LIN {X 0,Y 354.901,Z 540.274,A -85,B 0,C 180,E1 -13338.472,E2 -13338.472} C_VEL
LIN {X 0,Y 354.832,Z 540.28,A -85,B 0,C 180,E1 -13342.106,E2 -13342.106} C_VEL
LIN {X 0,Y 354.892,Z 540.272,A -85,B 0,C 180,E1 -13345.828,E2 -13345.828} C_VEL
LIN {X 0,Y 354.811,Z 540.288,A -85,B 0,C 180,E1 -13349.683,E2 -13349.683} C_VEL
LIN {X 0,Y 354.8,Z 540.289,A -85,B 0,C 180,E1 -13353.703,E2 -13353.703} C_VEL
LIN {X 0,Y 354.793,Z 540.268,A -85,B 0,C 180,E1 -13356.46,E2 -13356.46} C_VEL
LIN {X 0,Y 354.818,Z 540.287,A -85,B 0,C 180,E1 -13359.425,E2 -13359.425} C_VEL
LIN {X 0,Y 354.786,Z 540.277,A -85,B 0,C 180,E1 -13362.869,E2 -13362.869} C_VEL
LIN {X 0,Y 354.836,Z 540.279,A -85,B 0,C 180,E1 -13366.116,E2 -13366.116} C_VEL
LIN {X 0,Y 354.852,Z 540.284,A -85,B 0,C 180,E1 -13369.19,E2 -13369.19} C_VEL
LIN {X 0,Y 354.806,Z 540.261,A -85,B 0,C 180,E1 -13372.403,E2 -13372.403} C_VEL
LIN {X 0,Y 354.81,Z 540.29,A -85,B 0,C 180,E1 -13374.942,E2 -13374.942} C_VEL
LIN {X 0,Y 354.786,Z 540.225,A -85,B 0,C 180,E1 -13378.407,E2 -13378.407} C_VEL
LIN {X 0,Y 354.906,Z 540.442,A -85,B 0,C 180,E1 -13379.59,E2 -13379.59} C_VEL
LIN {X 0,Y 357.393,Z 551.805,A -85,B 0,C 180,E1 -13382.738,E2 -13382.738} C_VEL
LIN {X 0,Y 358.906,Z 560.837,A -85,B 0,C 180,E1 -13385.103,E2 -13385.103} C_VEL
LIN {X 0,Y 357.939,Z 570.577,A -85,B 0,C 180,E1 -13387.413,E2 -13387.413} C_VEL
LIN {X 0,Y 358.417,Z 573.829,A -85,B 0,C 180,E1 -13387.578,E2 -13387.578} C_VEL
LIN {X 0,Y 362.722,Z 599.14,A -85,B 0,C 180,E1 -13388.384,E2 -13388.384} C_VEL
LIN {X 0,Y 363.59,Z 605.924,A -85,B 0,C 180,E1 -13388.579,E2 -13388.579} C_VEL
LIN {X 0,Y 362.337,Z 679.031,A -85,B 0,C 180,E1 -13390.048,E2 -13390.048} C_VEL
LIN {X 0,Y 361.614,Z 692.225,A -85,B 0,C 180,E1 -13390.524,E2 -13390.524} C_VEL
LIN {X 0,Y 360.674,Z 705.472,A -85,B 0,C 180,E1 -13391.247,E2 -13391.247} C_VEL
LIN {X 0,Y 359.694,Z 716.606,A -85,B 0,C 180,E1 -13392.078,E2 -13392.078} C_VEL
LIN {X 0,Y 358.499,Z 728.189,A -85,B 0,C 180,E1 -13393.194,E2 -13393.194} C_VEL
LIN {X 0,Y 357.335,Z 739.084,A -85,B 0,C 180,E1 -13394.521,E2 -13394.521} C_VEL
LIN {X 0,Y 356.269,Z 748.832,A -85,B 0,C 180,E1 -13396.017,E2 -13396.017} C_VEL
LIN {X 0,Y 355.153,Z 757.764,A -85,B 0,C 180,E1 -13397.719,E2 -13397.719} C_VEL
LIN {X 0,Y 354.392,Z 764.959,A -85,B 0,C 180,E1 -13399.431,E2 -13399.431} C_VEL
LIN {X 0,Y 353.9,Z 769.814,A -85,B 0,C 180,E1 -13400.86,E2 -13400.86} C_VEL
LIN {X 0,Y 353.519,Z 774.536,A -85,B 0,C 180,E1 -13402.576,E2 -13402.576} C_VEL
LIN {X 0,Y 353.281,Z 778.149,A -85,B 0,C 180,E1 -13404.293,E2 -13404.293} C_VEL
LIN {X 0,Y 353.28,Z 780.014,A -85,B 0,C 180,E1 -13405.437,E2 -13405.437} C_VEL
LIN {X 0,Y 353.223,Z 781.409,A -85,B 0,C 180,E1 -13406.579,E2 -13406.579} C_VEL
LIN {X 0,Y 353.207,Z 784.384,A -85,B 0,C 180,E1 -13410.001,E2 -13410.001} C_VEL
LIN {X 0,Y 353.167,Z 784.671,A -85,B 0,C 180,E1 -13411.141,E2 -13411.141} C_VEL
LIN {X 0,Y 353.169,Z 784.334,A -85,B 0,C 180,E1 -13412.282,E2 -13412.282} C_VEL
LIN {X 0,Y 353.227,Z 783.434,A -85,B 0,C 180,E1 -13413.423,E2 -13413.423} C_VEL
LIN {X 0,Y 353.326,Z 781.996,A -85,B 0,C 180,E1 -13414.564,E2 -13414.564} C_VEL
LIN {X 0,Y 353.389,Z 779.211,A -85,B 0,C 180,E1 -13416.08,E2 -13416.08} C_VEL
LIN {X 0,Y 353.573,Z 775.814,A -85,B 0,C 180,E1 -13417.424,E2 -13417.424} C_VEL
LIN {X 0,Y 353.842,Z 771.158,A -85,B 0,C 180,E1 -13418.856,E2 -13418.856} C_VEL
LIN {X 0,Y 354.693,Z 761.5,A -85,B 0,C 180,E1 -13421.429,E2 -13421.429} C_VEL
LIN {X 0,Y 355.674,Z 753.468,A -85,B 0,C 180,E1 -13423.135,E2 -13423.135} C_VEL
LIN {X 0,Y 356.598,Z 745.28,A -85,B 0,C 180,E1 -13424.554,E2 -13424.554} C_VEL
LIN {X 0,Y 357.676,Z 735.298,A -85,B 0,C 180,E1 -13425.968,E2 -13425.968} C_VEL
LIN {X 0,Y 358.897,Z 724.022,A -85,B 0,C 180,E1 -13427.229,E2 -13427.229} C_VEL
LIN {X 0,Y 360.015,Z 712.981,A -85,B 0,C 180,E1 -13428.201,E2 -13428.201} C_VEL
LIN {X 0,Y 361.046,Z 700.746,A -85,B 0,C 180,E1 -13429.03,E2 -13429.03} C_VEL
LIN {X 0,Y 361.873,Z 687.862,A -85,B 0,C 180,E1 -13429.648,E2 -13429.648} C_VEL
LIN {X 0,Y 362.44,Z 674.152,A -85,B 0,C 180,E1 -13430.059,E2 -13430.059} C_VEL
LIN {X 0,Y 363.424,Z 603.753,A -85,B 0,C 180,E1 -13431.463,E2 -13431.463} C_VEL
LIN {X 0,Y 360.212,Z 583.434,A -85,B 0,C 180,E1 -13432.106,E2 -13432.106} C_VEL
LIN {X 0,Y 360.059,Z 575.5,A -85,B 0,C 180,E1 -13432.861,E2 -13432.861} C_VEL
LIN {X 0,Y 358.8,Z 563.274,A -85,B 0,C 180,E1 -13434.367,E2 -13434.367} C_VEL
LIN {X 0,Y 358.792,Z 559.513,A -85,B 0,C 180,E1 -13435.217,E2 -13435.217} C_VEL
LIN {X 0,Y 356.679,Z 548.182,A -85,B 0,C 180,E1 -13438.223,E2 -13438.223} C_VEL
LIN {X 0,Y 354.865,Z 540.354,A -85,B 0,C 180,E1 -13440.457,E2 -13440.457} C_VEL
LIN {X 0,Y 354.81,Z 540.287,A -85,B 0,C 180,E1 -13443.702,E2 -13443.702} C_VEL
LIN {X 0,Y 354.802,Z 540.289,A -85,B 0,C 180,E1 -13446.46,E2 -13446.46} C_VEL
LIN {X 0,Y 354.828,Z 540.287,A -85,B 0,C 180,E1 -13449.424,E2 -13449.424} C_VEL
LIN {X 0,Y 354.792,Z 540.29,A -85,B 0,C 180,E1 -13452.868,E2 -13452.868} C_VEL
LIN {X 0,Y 354.77,Z 540.292,A -85,B 0,C 180,E1 -13456.104,E2 -13456.104} C_VEL
LIN {X 0,Y 354.792,Z 540.289,A -85,B 0,C 180,E1 -13459.179,E2 -13459.179} C_VEL
LIN {X 0,Y 354.842,Z 540.398,A -85,B 0,C 180,E1 -13462.926,E2 -13462.926} C_VEL
LIN {X 0,Y 355.958,Z 543.292,A -85,B 0,C 180,E1 -13464.048,E2 -13464.048} C_VEL
LIN {X 0,Y 358.456,Z 549.807,A -85,B 0,C 180,E1 -13466.177,E2 -13466.177} C_VEL
LIN {X 0,Y 361.129,Z 558.129,A -85,B 0,C 180,E1 -13468.551,E2 -13468.551} C_VEL
LIN {X 0,Y 363.277,Z 567.144,A -85,B 0,C 180,E1 -13470.841,E2 -13470.841} C_VEL
LIN {X 0,Y 363.881,Z 571.171,A -85,B 0,C 180,E1 -13471.758,E2 -13471.758} C_VEL
LIN {X 0,Y 362.957,Z 580.6,A -85,B 0,C 180,E1 -13473.554,E2 -13473.554} C_VEL
LIN {X 0,Y 361.094,Z 599.26,A -85,B 0,C 180,E1 -13477.091,E2 -13477.091} C_VEL
LIN {X 0,Y 359.585,Z 617.559,A -85,B 0,C 180,E1 -13480.46,E2 -13480.46} C_VEL
LIN {X 0,Y 362.327,Z 632.262,A -85,B 0,C 180,E1 -13481.252,E2 -13481.252} C_VEL
LIN {X 0,Y 363.24,Z 640.661,A -85,B 0,C 180,E1 -13481.617,E2 -13481.617} C_VEL
LIN {X 0,Y 360.859,Z 699.458,A -85,B 0,C 180,E1 -13483.378,E2 -13483.378} C_VEL
LIN {X 0,Y 360.163,Z 709.923,A -85,B 0,C 180,E1 -13483.855,E2 -13483.855} C_VEL
LIN {X 0,Y 359.446,Z 720.79,A -85,B 0,C 180,E1 -13484.55,E2 -13484.55} C_VEL
LIN {X 0,Y 358.588,Z 730.488,A -85,B 0,C 180,E1 -13485.384,E2 -13485.384} C_VEL
LIN {X 0,Y 357.615,Z 739.515,A -85,B 0,C 180,E1 -13486.36,E2 -13486.36} C_VEL
LIN {X 0,Y 356.754,Z 747.891,A -85,B 0,C 180,E1 -13487.485,E2 -13487.485} C_VEL
LIN {X 0,Y 355.858,Z 756.225,A -85,B 0,C 180,E1 -13488.898,E2 -13488.898} C_VEL
LIN {X 0,Y 355.005,Z 762.802,A -85,B 0,C 180,E1 -13490.313,E2 -13490.313} C_VEL
LIN {X 0,Y 354.501,Z 767.137,A -85,B 0,C 180,E1 -13491.449,E2 -13491.449} C_VEL
LIN {X 0,Y 354.019,Z 771.909,A -85,B 0,C 180,E1 -13493.031,E2 -13493.031} C_VEL
LIN {X 0,Y 353.804,Z 774.792,A -85,B 0,C 180,E1 -13494.3,E2 -13494.3} C_VEL
LIN {X 0,Y 353.489,Z 776.752,A -85,B 0,C 180,E1 -13495.439,E2 -13495.439} C_VEL
LIN {X 0,Y 353.296,Z 778.158,A -85,B 0,C 180,E1 -13496.579,E2 -13496.579} C_VEL
LIN {X 0,Y 353.211,Z 779.033,A -85,B 0,C 180,E1 -13497.719,E2 -13497.719} C_VEL
LIN {X 0,Y 353.165,Z 779.34,A -85,B 0,C 180,E1 -13498.86,E2 -13498.86} C_VEL
LIN {X 0,Y 353.174,Z 779.041,A -85,B 0,C 180,E1 -13500,E2 -13500} C_VEL
LIN {X 0,Y 353.158,Z 778.209,A -85,B 0,C 180,E1 -13501.14,E2 -13501.14} C_VEL
LIN {X 0,Y 353.181,Z 776.838,A -85,B 0,C 180,E1 -13502.281,E2 -13502.281} C_VEL
LIN {X 0,Y 353.348,Z 773.707,A -85,B 0,C 180,E1 -13503.992,E2 -13503.992} C_VEL
LIN {X 0,Y 353.451,Z 769.159,A -85,B 0,C 180,E1 -13505.706,E2 -13505.706} C_VEL
LIN {X 0,Y 353.752,Z 764.04,A -85,B 0,C 180,E1 -13507.133,E2 -13507.133} C_VEL
LIN {X 0,Y 353.938,Z 759.008,A -85,B 0,C 180,E1 -13508.277,E2 -13508.277} C_VEL
LIN {X 0,Y 354.29,Z 752.942,A -85,B 0,C 180,E1 -13509.419,E2 -13509.419} C_VEL
LIN {X 0,Y 354.719,Z 745.593,A -85,B 0,C 180,E1 -13510.56,E2 -13510.56} C_VEL
LIN {X 0,Y 355.216,Z 736.599,A -85,B 0,C 180,E1 -13511.701,E2 -13511.701} C_VEL
LIN {X 0,Y 355.821,Z 726.511,A -85,B 0,C 180,E1 -13512.694,E2 -13512.694} C_VEL
LIN {X 0,Y 356.24,Z 717.243,A -85,B 0,C 180,E1 -13513.404,E2 -13513.404} C_VEL
LIN {X 0,Y 356.538,Z 707.589,A -85,B 0,C 180,E1 -13513.973,E2 -13513.973} C_VEL
LIN {X 0,Y 356.953,Z 695.613,A -85,B 0,C 180,E1 -13514.466,E2 -13514.466} C_VEL
LIN {X 0,Y 357.953,Z 636.557,A -85,B 0,C 180,E1 -13516.028,E2 -13516.028} C_VEL
LIN {X 0,Y 356.048,Z 617.144,A -85,B 0,C 180,E1 -13516.632,E2 -13516.632} C_VEL
LIN {X 0,Y 356.832,Z 600.704,A -85,B 0,C 180,E1 -13519.562,E2 -13519.562} C_VEL
LIN {X 0,Y 358.029,Z 581.082,A -85,B 0,C 180,E1 -13523.116,E2 -13523.116} C_VEL
LIN {X 0,Y 359.095,Z 562.902,A -85,B 0,C 180,E1 -13526.425,E2 -13526.425} C_VEL
LIN {X 0,Y 358.505,Z 557.641,A -85,B 0,C 180,E1 -13527.429,E2 -13527.429} C_VEL
LIN {X 0,Y 355.305,Z 542.619,A -85,B 0,C 180,E1 -13530.406,E2 -13530.406} C_VEL
LIN {X 0,Y 354.856,Z 540.394,A -85,B 0,C 180,E1 -13530.902,E2 -13530.902} C_VEL
LIN {X 0,Y 354.816,Z 540.289,A -85,B 0,C 180,E1 -13535.059,E2 -13535.059} C_VEL
LIN {X 0,Y 354.814,Z 540.286,A -85,B 0,C 180,E1 -13537.882,E2 -13537.882} C_VEL
LIN {X 0,Y 354.79,Z 540.253,A -85,B 0,C 180,E1 -13541.171,E2 -13541.171} C_VEL
LIN {X 0,Y 354.767,Z 540.28,A -85,B 0,C 180,E1 -13544.506,E2 -13544.506} C_VEL
LIN {X 0,Y 354.798,Z 540.285,A -85,B 0,C 180,E1 -13547.662,E2 -13547.662} C_VEL
LIN {X 0,Y 354.819,Z 540.256,A -85,B 0,C 180,E1 -13550.666,E2 -13550.666} C_VEL
LIN {X 0,Y 354.826,Z 540.285,A -85,B 0,C 180,E1 -13554.3,E2 -13554.3} C_VEL
LIN {X 0,Y 354.791,Z 540.29,A -85,B 0,C 180,E1 -13557.666,E2 -13557.666} C_VEL
LIN {X 0,Y 354.851,Z 540.28,A -85,B 0,C 180,E1 -13561.618,E2 -13561.618} C_VEL
LIN {X 0,Y 354.938,Z 540.423,A -85,B 0,C 180,E1 -13563.859,E2 -13563.859} C_VEL
LIN {X 0,Y 356.824,Z 549.951,A -85,B 0,C 180,E1 -13566.801,E2 -13566.801} C_VEL
LIN {X 0,Y 357.319,Z 552.539,A -85,B 0,C 180,E1 -13567.484,E2 -13567.484} C_VEL
LIN {X 0,Y 360.175,Z 560.7,A -85,B 0,C 180,E1 -13567.881,E2 -13567.881} C_VEL
LIN {X 0,Y 363.978,Z 579.583,A -85,B 0,C 180,E1 -13568.52,E2 -13568.52} C_VEL
LIN {X 0,Y 362.543,Z 658.643,A -85,B 0,C 180,E1 -13570.095,E2 -13570.095} C_VEL
LIN {X 0,Y 362.059,Z 671.327,A -85,B 0,C 180,E1 -13570.547,E2 -13570.547} C_VEL
LIN {X 0,Y 361.211,Z 684.868,A -85,B 0,C 180,E1 -13571.274,E2 -13571.274} C_VEL
LIN {X 0,Y 360.315,Z 696.202,A -85,B 0,C 180,E1 -13572.108,E2 -13572.108} C_VEL
LIN {X 0,Y 359.184,Z 707.773,A -85,B 0,C 180,E1 -13573.215,E2 -13573.215} C_VEL
LIN {X 0,Y 358.249,Z 718.308,A -85,B 0,C 180,E1 -13574.496,E2 -13574.496} C_VEL
LIN {X 0,Y 357.199,Z 726.851,A -85,B 0,C 180,E1 -13575.762,E2 -13575.762} C_VEL
LIN {X 0,Y 356.221,Z 734.721,A -85,B 0,C 180,E1 -13577.175,E2 -13577.175} C_VEL
LIN {X 0,Y 355.29,Z 742.41,A -85,B 0,C 180,E1 -13578.879,E2 -13578.879} C_VEL
LIN {X 0,Y 354.406,Z 749.468,A -85,B 0,C 180,E1 -13580.871,E2 -13580.871} C_VEL
LIN {X 0,Y 353.946,Z 754.166,A -85,B 0,C 180,E1 -13582.584,E2 -13582.584} C_VEL
LIN {X 0,Y 353.676,Z 757.756,A -85,B 0,C 180,E1 -13584.297,E2 -13584.297} C_VEL
LIN {X 0,Y 353.497,Z 759.613,A -85,B 0,C 180,E1 -13585.438,E2 -13585.438} C_VEL
LIN {X 0,Y 353.34,Z 761.013,A -85,B 0,C 180,E1 -13586.578,E2 -13586.578} C_VEL
LIN {X 0,Y 353.256,Z 762.621,A -85,B 0,C 180,E1 -13588.859,E2 -13588.859} C_VEL
LIN {X 0,Y 353.265,Z 762.853,A -85,B 0,C 180,E1 -13589.999,E2 -13589.999} C_VEL
LIN {X 0,Y 353.256,Z 762.665,A -85,B 0,C 180,E1 -13591.139,E2 -13591.139} C_VEL
LIN {X 0,Y 353.334,Z 761.117,A -85,B 0,C 180,E1 -13593.42,E2 -13593.42} C_VEL
LIN {X 0,Y 353.49,Z 759.761,A -85,B 0,C 180,E1 -13594.56,E2 -13594.56} C_VEL
LIN {X 0,Y 353.814,Z 756.019,A -85,B 0,C 180,E1 -13596.695,E2 -13596.695} C_VEL
LIN {X 0,Y 354.2,Z 751.45,A -85,B 0,C 180,E1 -13598.557,E2 -13598.557} C_VEL
LIN {X 0,Y 355.015,Z 745.015,A -85,B 0,C 180,E1 -13600.55,E2 -13600.55} C_VEL
LIN {X 0,Y 355.74,Z 738.678,A -85,B 0,C 180,E1 -13602.095,E2 -13602.095} C_VEL
LIN {X 0,Y 355.481,Z 735.193,A -85,B 0,C 180,E1 -13602.864,E2 -13602.864} C_VEL
LIN {X 0,Y 353.491,Z 729.249,A -85,B 0,C 180,E1 -13604.108,E2 -13604.108} C_VEL
LIN {X 0,Y 351.566,Z 722.759,A -85,B 0,C 180,E1 -13605.284,E2 -13605.284} C_VEL
LIN {X 0,Y 351.399,Z 718.404,A -85,B 0,C 180,E1 -13605.933,E2 -13605.933} C_VEL
LIN {X 0,Y 352.412,Z 707.819,A -85,B 0,C 180,E1 -13607.24,E2 -13607.24} C_VEL
LIN {X 0,Y 353.608,Z 695.92,A -85,B 0,C 180,E1 -13608.391,E2 -13608.391} C_VEL
LIN {X 0,Y 354.725,Z 683.279,A -85,B 0,C 180,E1 -13609.305,E2 -13609.305} C_VEL
LIN {X 0,Y 355.479,Z 670.635,A -85,B 0,C 180,E1 -13609.977,E2 -13609.977} C_VEL
LIN {X 0,Y 355.945,Z 658.621,A -85,B 0,C 180,E1 -13610.401,E2 -13610.401} C_VEL
LIN {X 0,Y 357.347,Z 579.911,A -85,B 0,C 180,E1 -13612.002,E2 -13612.002} C_VEL
LIN {X 0,Y 353.421,Z 561.513,A -85,B 0,C 180,E1 -13612.658,E2 -13612.658} C_VEL
LIN {X 0,Y 350.203,Z 552.682,A -85,B 0,C 180,E1 -13613.115,E2 -13613.115} C_VEL
LIN {X 0,Y 348.907,Z 546.369,A -85,B 0,C 180,E1 -13614.983,E2 -13614.983} C_VEL
LIN {X 0,Y 347.866,Z 541.204,A -85,B 0,C 180,E1 -13616.687,E2 -13616.687} C_VEL
LIN {X 0,Y 347.747,Z 541.157,A -85,B 0,C 180,E1 -13620.347,E2 -13620.347} C_VEL
LIN {X 0,Y 347.746,Z 541.17,A -85,B 0,C 180,E1 -13624.043,E2 -13624.043} C_VEL
LIN {X 0,Y 347.763,Z 541.166,A -85,B 0,C 180,E1 -13627.319,E2 -13627.319} C_VEL
LIN {X 0,Y 347.74,Z 541.16,A -85,B 0,C 180,E1 -13630.294,E2 -13630.294} C_VEL
LIN {X 0,Y 347.72,Z 541.166,A -85,B 0,C 180,E1 -13633.407,E2 -13633.407} C_VEL
LIN {X 0,Y 347.742,Z 541.163,A -85,B 0,C 180,E1 -13636.681,E2 -13636.681} C_VEL
LIN {X 0,Y 347.753,Z 541.153,A -85,B 0,C 180,E1 -13640.17,E2 -13640.17} C_VEL
LIN {X 0,Y 347.762,Z 541.151,A -85,B 0,C 180,E1 -13642.679,E2 -13642.679} C_VEL
LIN {X 0,Y 347.743,Z 541.167,A -85,B 0,C 180,E1 -13645.955,E2 -13645.955} C_VEL
LIN {X 0,Y 347.758,Z 541.169,A -85,B 0,C 180,E1 -13649.653,E2 -13649.653} C_VEL
LIN {X 0,Y 347.846,Z 541.145,A -85,B 0,C 180,E1 -13652.744,E2 -13652.744} C_VEL
LIN {X 0,Y 347.782,Z 541.159,A -85,B 0,C 180,E1 -13656.161,E2 -13656.161} C_VEL
LIN {X 0,Y 347.811,Z 541.159,A -85,B 0,C 180,E1 -13659.909,E2 -13659.909} C_VEL
LIN {X 0,Y 347.859,Z 541.147,A -85,B 0,C 180,E1 -13662.359,E2 -13662.359} C_VEL
LIN {X 0,Y 347.89,Z 541.149,A -85,B 0,C 180,E1 -13665.97,E2 -13665.97} C_VEL
LIN {X 0,Y 347.921,Z 541.135,A -85,B 0,C 180,E1 -13669.525,E2 -13669.525} C_VEL
LIN {X 0,Y 348.067,Z 541.126,A -85,B 0,C 180,E1 -13671.874,E2 -13671.874} C_VEL
LIN {X 0,Y 348.06,Z 541.126,A -85,B 0,C 180,E1 -13674.205,E2 -13674.205} C_VEL
LIN {X 0,Y 348.201,Z 541.102,A -85,B 0,C 180,E1 -13677.686,E2 -13677.686} C_VEL
LIN {X 0,Y 348.361,Z 541.091,A -85,B 0,C 180,E1 -13680,E2 -13680} C_VEL
LIN {X 0,Y 348.201,Z 541.103,A -85,B 0,C 180,E1 -13682.313,E2 -13682.313} C_VEL
LIN {X 0,Y 348.101,Z 541.122,A -85,B 0,C 180,E1 -13686.958,E2 -13686.958} C_VEL
LIN {X 0,Y 347.961,Z 541.134,A -85,B 0,C 180,E1 -13689.299,E2 -13689.299} C_VEL
LIN {X 0,Y 347.886,Z 541.148,A -85,B 0,C 180,E1 -13692.84,E2 -13692.84} C_VEL
LIN {X 0,Y 347.832,Z 541.147,A -85,B 0,C 180,E1 -13696.432,E2 -13696.432} C_VEL
LIN {X 0,Y 347.852,Z 541.153,A -85,B 0,C 180,E1 -13698.86,E2 -13698.86} C_VEL
LIN {X 0,Y 347.77,Z 541.159,A -85,B 0,C 180,E1 -13702.58,E2 -13702.58} C_VEL
LIN {X 0,Y 347.806,Z 541.16,A -85,B 0,C 180,E1 -13705.109,E2 -13705.109} C_VEL
LIN {X 0,Y 347.801,Z 541.158,A -85,B 0,C 180,E1 -13707.695,E2 -13707.695} C_VEL
LIN {X 0,Y 347.743,Z 541.163,A -85,B 0,C 180,E1 -13710.349,E2 -13710.349} C_VEL
LIN {X 0,Y 347.742,Z 541.165,A -85,B 0,C 180,E1 -13714.045,E2 -13714.045} C_VEL
LIN {X 0,Y 347.757,Z 541.148,A -85,B 0,C 180,E1 -13717.322,E2 -13717.322} C_VEL
LIN {X 0,Y 347.728,Z 541.169,A -85,B 0,C 180,E1 -13720.298,E2 -13720.298} C_VEL
LIN {X 0,Y 347.742,Z 541.158,A -85,B 0,C 180,E1 -13723.405,E2 -13723.405} C_VEL
LIN {X 0,Y 347.778,Z 541.155,A -85,B 0,C 180,E1 -13726.677,E2 -13726.677} C_VEL
LIN {X 0,Y 347.782,Z 541.157,A -85,B 0,C 180,E1 -13730.166,E2 -13730.166} C_VEL
LIN {X 0,Y 347.786,Z 541.158,A -85,B 0,C 180,E1 -13734.126,E2 -13734.126} C_VEL
LIN {X 0,Y 347.732,Z 541.104,A -85,B 0,C 180,E1 -13738.088,E2 -13738.088} C_VEL
LIN {X 0,Y 347.806,Z 541.332,A -85,B 0,C 180,E1 -13739.197,E2 -13739.197} C_VEL
LIN {X 0,Y 350.44,Z 553.084,A -85,B 0,C 180,E1 -13742.533,E2 -13742.533} C_VEL
LIN {X 0,Y 351.969,Z 561.98,A -85,B 0,C 180,E1 -13744.92,E2 -13744.92} C_VEL
LIN {X 0,Y 351.14,Z 570.571,A -85,B 0,C 180,E1 -13746.977,E2 -13746.977} C_VEL
LIN {X 0,Y 352.793,Z 579.779,A -85,B 0,C 180,E1 -13747.333,E2 -13747.333} C_VEL
LIN {X 0,Y 356.961,Z 605.801,A -85,B 0,C 180,E1 -13748.162,E2 -13748.162} C_VEL
LIN {X 0,Y 355.687,Z 678.839,A -85,B 0,C 180,E1 -13749.659,E2 -13749.659} C_VEL
LIN {X 0,Y 354.941,Z 692.03,A -85,B 0,C 180,E1 -13750.142,E2 -13750.142} C_VEL
LIN {X 0,Y 353.972,Z 705.273,A -85,B 0,C 180,E1 -13750.878,E2 -13750.878} C_VEL
LIN {X 0,Y 352.931,Z 716.405,A -85,B 0,C 180,E1 -13751.723,E2 -13751.723} C_VEL
LIN {X 0,Y 351.685,Z 727.987,A -85,B 0,C 180,E1 -13752.858,E2 -13752.858} C_VEL
LIN {X 0,Y 350.454,Z 738.96,A -85,B 0,C 180,E1 -13754.22,E2 -13754.22} C_VEL
LIN {X 0,Y 349.343,Z 748.628,A -85,B 0,C 180,E1 -13755.734,E2 -13755.734} C_VEL
LIN {X 0,Y 348.199,Z 757.561,A -85,B 0,C 180,E1 -13757.47,E2 -13757.47} C_VEL
LIN {X 0,Y 347.398,Z 764.755,A -85,B 0,C 180,E1 -13759.216,E2 -13759.216} C_VEL
LIN {X 0,Y 346.719,Z 771.305,A -85,B 0,C 180,E1 -13761.257,E2 -13761.257} C_VEL
LIN {X 0,Y 346.343,Z 775.644,A -85,B 0,C 180,E1 -13763.008,E2 -13763.008} C_VEL
LIN {X 0,Y 346.2,Z 777.944,A -85,B 0,C 180,E1 -13764.175,E2 -13764.175} C_VEL
LIN {X 0,Y 346.175,Z 779.809,A -85,B 0,C 180,E1 -13765.343,E2 -13765.343} C_VEL
LIN {X 0,Y 346.147,Z 781.205,A -85,B 0,C 180,E1 -13766.509,E2 -13766.509} C_VEL
LIN {X 0,Y 346.108,Z 784.272,A -85,B 0,C 180,E1 -13770.001,E2 -13770.001} C_VEL
LIN {X 0,Y 346.069,Z 784.599,A -85,B 0,C 180,E1 -13771.165,E2 -13771.165} C_VEL
LIN {X 0,Y 346.081,Z 784.321,A -85,B 0,C 180,E1 -13772.329,E2 -13772.329} C_VEL
LIN {X 0,Y 346.154,Z 783.509,A -85,B 0,C 180,E1 -13773.493,E2 -13773.493} C_VEL
LIN {X 0,Y 346.239,Z 782.157,A -85,B 0,C 180,E1 -13774.658,E2 -13774.658} C_VEL
LIN {X 0,Y 346.326,Z 779.703,A -85,B 0,C 180,E1 -13776.087,E2 -13776.087} C_VEL
LIN {X 0,Y 346.545,Z 776.182,A -85,B 0,C 180,E1 -13777.576,E2 -13777.576} C_VEL
LIN {X 0,Y 346.788,Z 772.656,A -85,B 0,C 180,E1 -13778.743,E2 -13778.743} C_VEL
LIN {X 0,Y 347.163,Z 767.179,A -85,B 0,C 180,E1 -13780.204,E2 -13780.204} C_VEL
LIN {X 0,Y 348.199,Z 757.494,A -85,B 0,C 180,E1 -13782.532,E2 -13782.532} C_VEL
LIN {X 0,Y 349.322,Z 748.545,A -85,B 0,C 180,E1 -13784.269,E2 -13784.269} C_VEL
LIN {X 0,Y 350.431,Z 738.64,A -85,B 0,C 180,E1 -13785.813,E2 -13785.813} C_VEL
LIN {X 0,Y 351.633,Z 727.851,A -85,B 0,C 180,E1 -13787.147,E2 -13787.147} C_VEL
LIN {X 0,Y 352.906,Z 716.238,A -85,B 0,C 180,E1 -13788.281,E2 -13788.281} C_VEL
LIN {X 0,Y 354.038,Z 703.927,A -85,B 0,C 180,E1 -13789.196,E2 -13789.196} C_VEL
LIN {X 0,Y 354.969,Z 690.954,A -85,B 0,C 180,E1 -13789.896,E2 -13789.896} C_VEL
LIN {X 0,Y 355.681,Z 678.349,A -85,B 0,C 180,E1 -13790.344,E2 -13790.344} C_VEL
LIN {X 0,Y 356.835,Z 604.804,A -85,B 0,C 180,E1 -13791.852,E2 -13791.852} C_VEL
LIN {X 0,Y 354.448,Z 588.941,A -85,B 0,C 180,E1 -13792.364,E2 -13792.364} C_VEL
LIN {X 0,Y 354.5,Z 578.627,A -85,B 0,C 180,E1 -13793.361,E2 -13793.361} C_VEL
LIN {X 0,Y 353.313,Z 565.845,A -85,B 0,C 180,E1 -13794.979,E2 -13794.979} C_VEL
LIN {X 0,Y 351.074,Z 556.144,A -85,B 0,C 180,E1 -13796.711,E2 -13796.711} C_VEL
LIN {X 0,Y 349.591,Z 548.971,A -85,B 0,C 180,E1 -13798.587,E2 -13798.587} C_VEL
LIN {X 0,Y 347.804,Z 541.258,A -85,B 0,C 180,E1 -13800.848,E2 -13800.848} C_VEL
LIN {X 0,Y 347.748,Z 541.169,A -85,B 0,C 180,E1 -13804.464,E2 -13804.464} C_VEL
LIN {X 0,Y 347.777,Z 541.166,A -85,B 0,C 180,E1 -13807.989,E2 -13807.989} C_VEL
LIN {X 0,Y 347.754,Z 541.167,A -85,B 0,C 180,E1 -13811.831,E2 -13811.831} C_VEL
LIN {X 0,Y 347.709,Z 541.175,A -85,B 0,C 180,E1 -13815.027,E2 -13815.027} C_VEL
LIN {X 0,Y 347.754,Z 541.168,A -85,B 0,C 180,E1 -13818.398,E2 -13818.398} C_VEL
LIN {X 0,Y 347.787,Z 541.37,A -85,B 0,C 180,E1 -13821.325,E2 -13821.325} C_VEL
LIN {X 0,Y 348.698,Z 543.886,A -85,B 0,C 180,E1 -13822.392,E2 -13822.392} C_VEL
LIN {X 0,Y 349.391,Z 544.951,A -85,B 0,C 180,E1 -13822.883,E2 -13822.883} C_VEL
LIN {X 0,Y 352.197,Z 552.266,A -85,B 0,C 180,E1 -13825.492,E2 -13825.492} C_VEL
LIN {X 0,Y 354.798,Z 560.426,A -85,B 0,C 180,E1 -13827.979,E2 -13827.979} C_VEL
LIN {X 0,Y 356.732,Z 568.33,A -85,B 0,C 180,E1 -13830.095,E2 -13830.095} C_VEL
LIN {X 0,Y 357.593,Z 574.274,A -85,B 0,C 180,E1 -13831.536,E2 -13831.536} C_VEL
LIN {X 0,Y 355.71,Z 591.496,A -85,B 0,C 180,E1 -13834.863,E2 -13834.863} C_VEL
LIN {X 0,Y 353.484,Z 613.273,A -85,B 0,C 180,E1 -13839.03,E2 -13839.03} C_VEL
LIN {X 0,Y 353.182,Z 617.698,A -85,B 0,C 180,E1 -13839.815,E2 -13839.815} C_VEL
LIN {X 0,Y 356.187,Z 633.43,A -85,B 0,C 180,E1 -13840.71,E2 -13840.71} C_VEL
LIN {X 0,Y 357.042,Z 641.425,A -85,B 0,C 180,E1 -13841.084,E2 -13841.084} C_VEL
LIN {X 0,Y 354.464,Z 699.698,A -85,B 0,C 180,E1 -13842.884,E2 -13842.884} C_VEL
LIN {X 0,Y 353.79,Z 709.378,A -85,B 0,C 180,E1 -13843.334,E2 -13843.334} C_VEL
LIN {X 0,Y 352.925,Z 721.212,A -85,B 0,C 180,E1 -13844.109,E2 -13844.109} C_VEL
LIN {X 0,Y 351.981,Z 730.75,A -85,B 0,C 180,E1 -13844.955,E2 -13844.955} C_VEL
LIN {X 0,Y 350.956,Z 739.685,A -85,B 0,C 180,E1 -13845.948,E2 -13845.948} C_VEL
LIN {X 0,Y 350.109,Z 747.08,A -85,B 0,C 180,E1 -13846.948,E2 -13846.948} C_VEL
LIN {X 0,Y 349.148,Z 755.674,A -85,B 0,C 180,E1 -13848.388,E2 -13848.388} C_VEL
LIN {X 0,Y 348.212,Z 762.369,A -85,B 0,C 180,E1 -13849.828,E2 -13849.828} C_VEL
LIN {X 0,Y 347.524,Z 767.736,A -85,B 0,C 180,E1 -13851.276,E2 -13851.276} C_VEL
LIN {X 0,Y 347.123,Z 771.195,A -85,B 0,C 180,E1 -13852.438,E2 -13852.438} C_VEL
LIN {X 0,Y 346.766,Z 775.162,A -85,B 0,C 180,E1 -13854.184,E2 -13854.184} C_VEL
LIN {X 0,Y 346.439,Z 777.035,A -85,B 0,C 180,E1 -13855.346,E2 -13855.346} C_VEL
LIN {X 0,Y 346.224,Z 778.353,A -85,B 0,C 180,E1 -13856.509,E2 -13856.509} C_VEL
LIN {X 0,Y 346.123,Z 779.14,A -85,B 0,C 180,E1 -13857.673,E2 -13857.673} C_VEL
LIN {X 0,Y 346.068,Z 779.396,A -85,B 0,C 180,E1 -13858.836,E2 -13858.836} C_VEL
LIN {X 0,Y 346.074,Z 779.051,A -85,B 0,C 180,E1 -13860,E2 -13860} C_VEL
LIN {X 0,Y 346.061,Z 778.124,A -85,B 0,C 180,E1 -13861.164,E2 -13861.164} C_VEL
LIN {X 0,Y 346.127,Z 775.788,A -85,B 0,C 180,E1 -13862.91,E2 -13862.91} C_VEL
LIN {X 0,Y 346.314,Z 771.991,A -85,B 0,C 180,E1 -13864.656,E2 -13864.656} C_VEL
LIN {X 0,Y 346.45,Z 767.166,A -85,B 0,C 180,E1 -13866.274,E2 -13866.274} C_VEL
LIN {X 0,Y 346.778,Z 761.051,A -85,B 0,C 180,E1 -13867.863,E2 -13867.863} C_VEL
LIN {X 0,Y 347.173,Z 753.767,A -85,B 0,C 180,E1 -13869.32,E2 -13869.32} C_VEL
LIN {X 0,Y 347.643,Z 745.538,A -85,B 0,C 180,E1 -13870.63,E2 -13870.63} C_VEL
LIN {X 0,Y 348.149,Z 736.517,A -85,B 0,C 180,E1 -13871.794,E2 -13871.794} C_VEL
LIN {X 0,Y 348.779,Z 726.368,A -85,B 0,C 180,E1 -13872.806,E2 -13872.806} C_VEL
LIN {X 0,Y 349.201,Z 717.059,A -85,B 0,C 180,E1 -13873.531,E2 -13873.531} C_VEL
LIN {X 0,Y 349.497,Z 707.355,A -85,B 0,C 180,E1 -13874.112,E2 -13874.112} C_VEL
LIN {X 0,Y 349.934,Z 695.198,A -85,B 0,C 180,E1 -13874.614,E2 -13874.614} C_VEL
LIN {X 0,Y 350.971,Z 637.15,A -85,B 0,C 180,E1 -13876.193,E2 -13876.193} C_VEL
LIN {X 0,Y 349.033,Z 617.196,A -85,B 0,C 180,E1 -13876.825,E2 -13876.825} C_VEL
LIN {X 0,Y 349.811,Z 601.182,A -85,B 0,C 180,E1 -13879.719,E2 -13879.719} C_VEL
LIN {X 0,Y 351.07,Z 581.28,A -85,B 0,C 180,E1 -13883.375,E2 -13883.375} C_VEL
LIN {X 0,Y 352.127,Z 563.318,A -85,B 0,C 180,E1 -13886.684,E2 -13886.684} C_VEL
LIN {X 0,Y 350.727,Z 554.833,A -85,B 0,C 180,E1 -13888.353,E2 -13888.353} C_VEL
LIN {X 0,Y 347.808,Z 541.27,A -85,B 0,C 180,E1 -13891.142,E2 -13891.142} C_VEL
LIN {X 0,Y 347.748,Z 541.168,A -85,B 0,C 180,E1 -13894.464,E2 -13894.464} C_VEL
LIN {X 0,Y 347.781,Z 541.162,A -85,B 0,C 180,E1 -13897.989,E2 -13897.989} C_VEL
LIN {X 0,Y 347.754,Z 541.122,A -85,B 0,C 180,E1 -13901.83,E2 -13901.83} C_VEL
LIN {X 0,Y 347.71,Z 541.162,A -85,B 0,C 180,E1 -13905.026,E2 -13905.026} C_VEL
LIN {X 0,Y 347.754,Z 541.157,A -85,B 0,C 180,E1 -13908.397,E2 -13908.397} C_VEL
LIN {X 0,Y 347.777,Z 541.152,A -85,B 0,C 180,E1 -13912.011,E2 -13912.011} C_VEL
LIN {X 0,Y 347.748,Z 541.158,A -85,B 0,C 180,E1 -13915.536,E2 -13915.536} C_VEL
LIN {X 0,Y 347.749,Z 541.164,A -85,B 0,C 180,E1 -13918.3,E2 -13918.3} C_VEL
LIN {X 0,Y 347.783,Z 541.162,A -85,B 0,C 180,E1 -13920.987,E2 -13920.987} C_VEL
LIN {X 0,Y 347.898,Z 541.271,A -85,B 0,C 180,E1 -13923.48,E2 -13923.48} C_VEL
LIN {X 0,Y 349.965,Z 551.705,A -85,B 0,C 180,E1 -13926.765,E2 -13926.765} C_VEL
LIN {X 0,Y 350.215,Z 552.951,A -85,B 0,C 180,E1 -13927.018,E2 -13927.018} C_VEL
LIN {X 0,Y 353.926,Z 563.388,A -85,B 0,C 180,E1 -13927.522,E2 -13927.522} C_VEL
LIN {X 0,Y 357.382,Z 580.666,A -85,B 0,C 180,E1 -13928.121,E2 -13928.121} C_VEL
LIN {X 0,Y 355.903,Z 658.865,A -85,B 0,C 180,E1 -13929.707,E2 -13929.707} C_VEL
LIN {X 0,Y 355.396,Z 671.542,A -85,B 0,C 180,E1 -13930.167,E2 -13930.167} C_VEL
LIN {X 0,Y 354.517,Z 685.08,A -85,B 0,C 180,E1 -13930.906,E2 -13930.906} C_VEL
LIN {X 0,Y 353.579,Z 696.412,A -85,B 0,C 180,E1 -13931.755,E2 -13931.755} C_VEL
LIN {X 0,Y 352.368,Z 708.321,A -85,B 0,C 180,E1 -13932.92,E2 -13932.92} C_VEL
LIN {X 0,Y 351.411,Z 718.516,A -85,B 0,C 180,E1 -13934.187,E2 -13934.187} C_VEL
LIN {X 0,Y 350.321,Z 727.059,A -85,B 0,C 180,E1 -13935.476,E2 -13935.476} C_VEL
LIN {X 0,Y 349.282,Z 734.929,A -85,B 0,C 180,E1 -13936.916,E2 -13936.916} C_VEL
LIN {X 0,Y 348.321,Z 742.616,A -85,B 0,C 180,E1 -13938.654,E2 -13938.654} C_VEL
LIN {X 0,Y 347.656,Z 747.865,A -85,B 0,C 180,E1 -13940.105,E2 -13940.105} C_VEL
LIN {X 0,Y 347.019,Z 752.957,A -85,B 0,C 180,E1 -13941.849,E2 -13941.849} C_VEL
LIN {X 0,Y 346.728,Z 756.326,A -85,B 0,C 180,E1 -13943.32,E2 -13943.32} C_VEL
LIN {X 0,Y 346.439,Z 759.818,A -85,B 0,C 180,E1 -13945.345,E2 -13945.345} C_VEL
LIN {X 0,Y 346.264,Z 761.218,A -85,B 0,C 180,E1 -13946.508,E2 -13946.508} C_VEL
LIN {X 0,Y 346.16,Z 762.826,A -85,B 0,C 180,E1 -13948.836,E2 -13948.836} C_VEL
LIN {X 0,Y 346.168,Z 763.058,A -85,B 0,C 180,E1 -13949.999,E2 -13949.999} C_VEL
LIN {X 0,Y 346.159,Z 762.869,A -85,B 0,C 180,E1 -13951.162,E2 -13951.162} C_VEL
LIN {X 0,Y 346.259,Z 761.321,A -85,B 0,C 180,E1 -13953.49,E2 -13953.49} C_VEL
LIN {X 0,Y 346.432,Z 759.964,A -85,B 0,C 180,E1 -13954.653,E2 -13954.653} C_VEL
LIN {X 0,Y 346.727,Z 756.547,A -85,B 0,C 180,E1 -13956.679,E2 -13956.679} C_VEL
LIN {X 0,Y 347.175,Z 751.654,A -85,B 0,C 180,E1 -13958.732,E2 -13958.732} C_VEL
LIN {X 0,Y 348.004,Z 745.219,A -85,B 0,C 180,E1 -13960.765,E2 -13960.765} C_VEL
LIN {X 0,Y 348.861,Z 738.146,A -85,B 0,C 180,E1 -13962.506,E2 -13962.506} C_VEL
LIN {X 0,Y 350.045,Z 729.329,A -85,B 0,C 180,E1 -13964.237,E2 -13964.237} C_VEL
LIN {X 0,Y 351.213,Z 720.287,A -85,B 0,C 180,E1 -13965.67,E2 -13965.67} C_VEL
LIN {X 0,Y 351.399,Z 718.404,A -85,B 0,C 180,E1 -13965.933,E2 -13965.933} C_VEL
LIN {X 0,Y 351.194,Z 713.945,A -85,B 0,C 180,E1 -13966.555,E2 -13966.555} C_VEL
LIN {X 0,Y 349.169,Z 706.484,A -85,B 0,C 180,E1 -13967.574,E2 -13967.574} C_VEL
LIN {X 0,Y 347.232,Z 698.604,A -85,B 0,C 180,E1 -13968.505,E2 -13968.505} C_VEL
LIN {X 0,Y 347.152,Z 693.415,A -85,B 0,C 180,E1 -13968.98,E2 -13968.98} C_VEL
LIN {X 0,Y 348.188,Z 681.217,A -85,B 0,C 180,E1 -13969.836,E2 -13969.836} C_VEL
LIN {X 0,Y 348.902,Z 668.23,A -85,B 0,C 180,E1 -13970.485,E2 -13970.485} C_VEL
LIN {X 0,Y 349.443,Z 654.312,A -85,B 0,C 180,E1 -13970.914,E2 -13970.914} C_VEL
LIN {X 0,Y 350.796,Z 581.032,A -85,B 0,C 180,E1 -13972.414,E2 -13972.414} C_VEL
LIN {X 0,Y 347.06,Z 563.54,A -85,B 0,C 180,E1 -13973.057,E2 -13973.057} C_VEL
LIN {X 0,Y 343.049,Z 552.944,A -85,B 0,C 180,E1 -13973.62,E2 -13973.62} C_VEL
LIN {X 0,Y 341.509,Z 545.362,A -85,B 0,C 180,E1 -13975.931,E2 -13975.931} C_VEL
LIN {X 0,Y 340.834,Z 542.049,A -85,B 0,C 180,E1 -13977.111,E2 -13977.111} C_VEL
LIN {X 0,Y 340.696,Z 542.044,A -85,B 0,C 180,E1 -13981.043,E2 -13981.043} C_VEL
LIN {X 0,Y 340.716,Z 542.04,A -85,B 0,C 180,E1 -13985.278,E2 -13985.278} C_VEL
LIN {X 0,Y 340.71,Z 542.043,A -85,B 0,C 180,E1 -13988.386,E2 -13988.386} C_VEL
LIN {X 0,Y 340.699,Z 542.046,A -85,B 0,C 180,E1 -13992.045,E2 -13992.045} C_VEL
LIN {X 0,Y 340.663,Z 542.045,A -85,B 0,C 180,E1 -13996.223,E2 -13996.223} C_VEL
LIN {X 0,Y 340.7,Z 542.044,A -85,B 0,C 180,E1 -13998.692,E2 -13998.692} C_VEL
LIN {X 0,Y 340.736,Z 542.019,A -85,B 0,C 180,E1 -14001.773,E2 -14001.773} C_VEL
LIN {X 0,Y 340.719,Z 542.045,A -85,B 0,C 180,E1 -14005.594,E2 -14005.594} C_VEL
LIN {X 0,Y 340.698,Z 542.043,A -85,B 0,C 180,E1 -14008.955,E2 -14008.955} C_VEL
LIN {X 0,Y 340.773,Z 542.025,A -85,B 0,C 180,E1 -14012.473,E2 -14012.473} C_VEL
LIN {X 0,Y 340.749,Z 542.039,A -85,B 0,C 180,E1 -14015.638,E2 -14015.638} C_VEL
LIN {X 0,Y 340.742,Z 542.037,A -85,B 0,C 180,E1 -14019.474,E2 -14019.474} C_VEL
LIN {X 0,Y 340.851,Z 542.021,A -85,B 0,C 180,E1 -14021.984,E2 -14021.984} C_VEL
LIN {X 0,Y 340.862,Z 542.024,A -85,B 0,C 180,E1 -14025.705,E2 -14025.705} C_VEL
LIN {X 0,Y 340.863,Z 542.016,A -85,B 0,C 180,E1 -14029.306,E2 -14029.306} C_VEL
LIN {X 0,Y 341.068,Z 541.997,A -85,B 0,C 180,E1 -14032.898,E2 -14032.898} C_VEL
LIN {X 0,Y 341.163,Z 541.977,A -85,B 0,C 180,E1 -14037.639,E2 -14037.639} C_VEL
LIN {X 0,Y 341.31,Z 541.97,A -85,B 0,C 180,E1 -14040,E2 -14040} C_VEL
LIN {X 0,Y 341.163,Z 541.979,A -85,B 0,C 180,E1 -14042.361,E2 -14042.361} C_VEL
LIN {X 0,Y 341.07,Z 541.999,A -85,B 0,C 180,E1 -14047.102,E2 -14047.102} C_VEL
LIN {X 0,Y 340.866,Z 542.013,A -85,B 0,C 180,E1 -14050.694,E2 -14050.694} C_VEL
LIN {X 0,Y 340.855,Z 542.022,A -85,B 0,C 180,E1 -14054.325,E2 -14054.325} C_VEL
LIN {X 0,Y 340.831,Z 542.027,A -85,B 0,C 180,E1 -14058.468,E2 -14058.468} C_VEL
LIN {X 0,Y 340.747,Z 542.033,A -85,B 0,C 180,E1 -14061.857,E2 -14061.857} C_VEL
LIN {X 0,Y 340.766,Z 542.034,A -85,B 0,C 180,E1 -14065.665,E2 -14065.665} C_VEL
LIN {X 0,Y 340.721,Z 542.042,A -85,B 0,C 180,E1 -14068.321,E2 -14068.321} C_VEL
LIN {X 0,Y 340.692,Z 542.041,A -85,B 0,C 180,E1 -14071.045,E2 -14071.045} C_VEL
LIN {X 0,Y 340.712,Z 542.032,A -85,B 0,C 180,E1 -14075.28,E2 -14075.28} C_VEL
LIN {X 0,Y 340.705,Z 542.042,A -85,B 0,C 180,E1 -14078.387,E2 -14078.387} C_VEL
LIN {X 0,Y 340.696,Z 542.032,A -85,B 0,C 180,E1 -14082.047,E2 -14082.047} C_VEL
LIN {X 0,Y 340.732,Z 542.043,A -85,B 0,C 180,E1 -14085.471,E2 -14085.471} C_VEL
LIN {X 0,Y 340.721,Z 542.043,A -85,B 0,C 180,E1 -14088.697,E2 -14088.697} C_VEL
LIN {X 0,Y 340.736,Z 542.013,A -85,B 0,C 180,E1 -14091.775,E2 -14091.775} C_VEL
LIN {X 0,Y 340.72,Z 542.037,A -85,B 0,C 180,E1 -14095.596,E2 -14095.596} C_VEL
LIN {X 0,Y 340.735,Z 542.067,A -85,B 0,C 180,E1 -14098.702,E2 -14098.702} C_VEL
LIN {X 0,Y 343.178,Z 552.874,A -85,B 0,C 180,E1 -14101.901,E2 -14101.901} C_VEL
LIN {X 0,Y 345.004,Z 562.916,A -85,B 0,C 180,E1 -14104.674,E2 -14104.674} C_VEL
LIN {X 0,Y 344.445,Z 569.18,A -85,B 0,C 180,E1 -14106.252,E2 -14106.252} C_VEL
LIN {X 0,Y 344.392,Z 570.811,A -85,B 0,C 180,E1 -14106.533,E2 -14106.533} C_VEL
LIN {X 0,Y 349.428,Z 599.922,A -85,B 0,C 180,E1 -14107.543,E2 -14107.543} C_VEL
LIN {X 0,Y 350.376,Z 608.08,A -85,B 0,C 180,E1 -14107.784,E2 -14107.784} C_VEL
LIN {X 0,Y 349.019,Z 678.647,A -85,B 0,C 180,E1 -14109.252,E2 -14109.252} C_VEL
LIN {X 0,Y 348.279,Z 691.834,A -85,B 0,C 180,E1 -14109.746,E2 -14109.746} C_VEL
LIN {X 0,Y 347.356,Z 703.958,A -85,B 0,C 180,E1 -14110.422,E2 -14110.422} C_VEL
LIN {X 0,Y 346.179,Z 716.205,A -85,B 0,C 180,E1 -14111.353,E2 -14111.353} C_VEL
LIN {X 0,Y 344.892,Z 727.786,A -85,B 0,C 180,E1 -14112.51,E2 -14112.51} C_VEL
LIN {X 0,Y 343.684,Z 737.768,A -85,B 0,C 180,E1 -14113.76,E2 -14113.76} C_VEL
LIN {X 0,Y 342.61,Z 746.748,A -85,B 0,C 180,E1 -14115.144,E2 -14115.144} C_VEL
LIN {X 0,Y 341.623,Z 754.621,A -85,B 0,C 180,E1 -14116.619,E2 -14116.619} C_VEL
LIN {X 0,Y 340.578,Z 762.31,A -85,B 0,C 180,E1 -14118.394,E2 -14118.394} C_VEL
LIN {X 0,Y 340.035,Z 767.584,A -85,B 0,C 180,E1 -14119.883,E2 -14119.883} C_VEL
LIN {X 0,Y 339.53,Z 772.693,A -85,B 0,C 180,E1 -14121.67,E2 -14121.67} C_VEL
LIN {X 0,Y 339.175,Z 776.665,A -85,B 0,C 180,E1 -14123.457,E2 -14123.457} C_VEL
LIN {X 0,Y 339.076,Z 779.604,A -85,B 0,C 180,E1 -14125.245,E2 -14125.245} C_VEL
LIN {X 0,Y 339.071,Z 781.001,A -85,B 0,C 180,E1 -14126.436,E2 -14126.436} C_VEL
LIN {X 0,Y 339.009,Z 784.126,A -85,B 0,C 180,E1 -14130.001,E2 -14130.001} C_VEL
LIN {X 0,Y 338.974,Z 784.495,A -85,B 0,C 180,E1 -14131.189,E2 -14131.189} C_VEL
LIN {X 0,Y 338.996,Z 784.308,A -85,B 0,C 180,E1 -14132.377,E2 -14132.377} C_VEL
LIN {X 0,Y 339.081,Z 783.595,A -85,B 0,C 180,E1 -14133.566,E2 -14133.566} C_VEL
LIN {X 0,Y 339.157,Z 782.349,A -85,B 0,C 180,E1 -14134.756,E2 -14134.756} C_VEL
LIN {X 0,Y 339.299,Z 779.347,A -85,B 0,C 180,E1 -14136.542,E2 -14136.542} C_VEL
LIN {X 0,Y 339.501,Z 776.595,A -85,B 0,C 180,E1 -14137.734,E2 -14137.734} C_VEL
LIN {X 0,Y 339.923,Z 771.184,A -85,B 0,C 180,E1 -14139.522,E2 -14139.522} C_VEL
LIN {X 0,Y 340.527,Z 764.035,A -85,B 0,C 180,E1 -14141.308,E2 -14141.308} C_VEL
LIN {X 0,Y 342.023,Z 751.562,A -85,B 0,C 180,E1 -14143.973,E2 -14143.973} C_VEL
LIN {X 0,Y 343.141,Z 742.462,A -85,B 0,C 180,E1 -14145.537,E2 -14145.537} C_VEL
LIN {X 0,Y 344.252,Z 732.562,A -85,B 0,C 180,E1 -14146.914,E2 -14146.914} C_VEL
LIN {X 0,Y 345.66,Z 720.745,A -85,B 0,C 180,E1 -14148.217,E2 -14148.217} C_VEL
LIN {X 0,Y 346.865,Z 708.86,A -85,B 0,C 180,E1 -14149.224,E2 -14149.224} C_VEL
LIN {X 0,Y 347.924,Z 696.492,A -85,B 0,C 180,E1 -14150.008,E2 -14150.008} C_VEL
LIN {X 0,Y 348.793,Z 683.763,A -85,B 0,C 180,E1 -14150.571,E2 -14150.571} C_VEL
LIN {X 0,Y 349.216,Z 670.353,A -85,B 0,C 180,E1 -14150.93,E2 -14150.93} C_VEL
LIN {X 0,Y 350.265,Z 605.79,A -85,B 0,C 180,E1 -14152.258,E2 -14152.258} C_VEL
LIN {X 0,Y 348.556,Z 594.193,A -85,B 0,C 180,E1 -14152.665,E2 -14152.665} C_VEL
LIN {X 0,Y 348.943,Z 581.232,A -85,B 0,C 180,E1 -14153.943,E2 -14153.943} C_VEL
LIN {X 0,Y 347.996,Z 569.147,A -85,B 0,C 180,E1 -14155.538,E2 -14155.538} C_VEL
LIN {X 0,Y 345.994,Z 560.149,A -85,B 0,C 180,E1 -14157.196,E2 -14157.196} C_VEL
LIN {X 0,Y 343.46,Z 550.924,A -85,B 0,C 180,E1 -14159.414,E2 -14159.414} C_VEL
LIN {X 0,Y 342.231,Z 545.739,A -85,B 0,C 180,E1 -14160.891,E2 -14160.891} C_VEL
LIN {X 0,Y 340.722,Z 542.311,A -85,B 0,C 180,E1 -14162.433,E2 -14162.433} C_VEL
LIN {X 0,Y 340.722,Z 542.041,A -85,B 0,C 180,E1 -14165.279,E2 -14165.279} C_VEL
LIN {X 0,Y 340.713,Z 542.043,A -85,B 0,C 180,E1 -14168.386,E2 -14168.386} C_VEL
LIN {X 0,Y 340.702,Z 542.044,A -85,B 0,C 180,E1 -14172.046,E2 -14172.046} C_VEL
LIN {X 0,Y 340.655,Z 542.05,A -85,B 0,C 180,E1 -14176.227,E2 -14176.227} C_VEL
LIN {X 0,Y 340.731,Z 542.305,A -85,B 0,C 180,E1 -14179.17,E2 -14179.17} C_VEL
LIN {X 0,Y 342.516,Z 546.143,A -85,B 0,C 180,E1 -14181.235,E2 -14181.235} C_VEL
LIN {X 0,Y 344.27,Z 550.421,A -85,B 0,C 180,E1 -14183.079,E2 -14183.079} C_VEL
LIN {X 0,Y 346.655,Z 556.725,A -85,B 0,C 180,E1 -14185.412,E2 -14185.412} C_VEL
LIN {X 0,Y 348.929,Z 564.19,A -85,B 0,C 180,E1 -14187.775,E2 -14187.775} C_VEL
LIN {X 0,Y 350.704,Z 571.968,A -85,B 0,C 180,E1 -14189.934,E2 -14189.934} C_VEL
LIN {X 0,Y 351.41,Z 577.689,A -85,B 0,C 180,E1 -14191.315,E2 -14191.315} C_VEL
LIN {X 0,Y 348.848,Z 598.345,A -85,B 0,C 180,E1 -14195.393,E2 -14195.393} C_VEL
LIN {X 0,Y 346.839,Z 617.57,A -85,B 0,C 180,E1 -14199.098,E2 -14199.098} C_VEL
LIN {X 0,Y 349.751,Z 632.37,A -85,B 0,C 180,E1 -14200.025,E2 -14200.025} C_VEL
LIN {X 0,Y 350.915,Z 642.636,A -85,B 0,C 180,E1 -14200.527,E2 -14200.527} C_VEL
LIN {X 0,Y 348.169,Z 699.221,A -85,B 0,C 180,E1 -14202.34,E2 -14202.34} C_VEL
LIN {X 0,Y 347.358,Z 710.159,A -85,B 0,C 180,E1 -14202.864,E2 -14202.864} C_VEL
LIN {X 0,Y 346.433,Z 721.773,A -85,B 0,C 180,E1 -14203.652,E2 -14203.652} C_VEL
LIN {X 0,Y 345.417,Z 731.216,A -85,B 0,C 180,E1 -14204.511,E2 -14204.511} C_VEL
LIN {X 0,Y 344.326,Z 740.097,A -85,B 0,C 180,E1 -14205.521,E2 -14205.521} C_VEL
LIN {X 0,Y 343.31,Z 748.367,A -85,B 0,C 180,E1 -14206.685,E2 -14206.685} C_VEL
LIN {X 0,Y 342.268,Z 756.568,A -85,B 0,C 180,E1 -14208.151,E2 -14208.151} C_VEL
LIN {X 0,Y 341.285,Z 763.116,A -85,B 0,C 180,E1 -14209.619,E2 -14209.619} C_VEL
LIN {X 0,Y 340.559,Z 768.376,A -85,B 0,C 180,E1 -14211.096,E2 -14211.096} C_VEL
LIN {X 0,Y 339.947,Z 773.302,A -85,B 0,C 180,E1 -14212.909,E2 -14212.909} C_VEL
LIN {X 0,Y 339.731,Z 775.586,A -85,B 0,C 180,E1 -14214.063,E2 -14214.063} C_VEL
LIN {X 0,Y 339.391,Z 777.345,A -85,B 0,C 180,E1 -14215.249,E2 -14215.249} C_VEL
LIN {X 0,Y 339.156,Z 778.56,A -85,B 0,C 180,E1 -14216.436,E2 -14216.436} C_VEL
LIN {X 0,Y 339.037,Z 779.248,A -85,B 0,C 180,E1 -14217.624,E2 -14217.624} C_VEL
LIN {X 0,Y 338.975,Z 779.418,A -85,B 0,C 180,E1 -14218.812,E2 -14218.812} C_VEL
LIN {X 0,Y 338.978,Z 779.032,A -85,B 0,C 180,E1 -14220,E2 -14220} C_VEL
LIN {X 0,Y 338.967,Z 778.034,A -85,B 0,C 180,E1 -14221.188,E2 -14221.188} C_VEL
LIN {X 0,Y 339.051,Z 775.523,A -85,B 0,C 180,E1 -14222.971,E2 -14222.971} C_VEL
LIN {X 0,Y 339.213,Z 773.105,A -85,B 0,C 180,E1 -14224.159,E2 -14224.159} C_VEL
LIN {X 0,Y 339.3,Z 768.132,A -85,B 0,C 180,E1 -14225.945,E2 -14225.945} C_VEL
LIN {X 0,Y 339.648,Z 762.751,A -85,B 0,C 180,E1 -14227.431,E2 -14227.431} C_VEL
LIN {X 0,Y 339.942,Z 755.991,A -85,B 0,C 180,E1 -14228.92,E2 -14228.92} C_VEL
LIN {X 0,Y 340.479,Z 747.348,A -85,B 0,C 180,E1 -14230.406,E2 -14230.406} C_VEL
LIN {X 0,Y 340.986,Z 738.671,A -85,B 0,C 180,E1 -14231.593,E2 -14231.593} C_VEL
LIN {X 0,Y 341.479,Z 729.273,A -85,B 0,C 180,E1 -14232.631,E2 -14232.631} C_VEL
LIN {X 0,Y 342.102,Z 717.734,A -85,B 0,C 180,E1 -14233.59,E2 -14233.59} C_VEL
LIN {X 0,Y 342.437,Z 708.281,A -85,B 0,C 180,E1 -14234.182,E2 -14234.182} C_VEL
LIN {X 0,Y 342.762,Z 697.708,A -85,B 0,C 180,E1 -14234.661,E2 -14234.661} C_VEL
LIN {X 0,Y 344.013,Z 638.495,A -85,B 0,C 180,E1 -14236.342,E2 -14236.342} C_VEL
LIN {X 0,Y 342.035,Z 617.257,A -85,B 0,C 180,E1 -14237.026,E2 -14237.026} C_VEL
LIN {X 0,Y 342.651,Z 604.473,A -85,B 0,C 180,E1 -14239.352,E2 -14239.352} C_VEL
LIN {X 0,Y 344.029,Z 583.073,A -85,B 0,C 180,E1 -14243.333,E2 -14243.333} C_VEL
LIN {X 0,Y 345.146,Z 565.504,A -85,B 0,C 180,E1 -14246.614,E2 -14246.614} C_VEL
LIN {X 0,Y 344.583,Z 560.215,A -85,B 0,C 180,E1 -14247.646,E2 -14247.646} C_VEL
LIN {X 0,Y 341.598,Z 546.21,A -85,B 0,C 180,E1 -14250.494,E2 -14250.494} C_VEL
LIN {X 0,Y 340.748,Z 542.153,A -85,B 0,C 180,E1 -14251.385,E2 -14251.385} C_VEL
LIN {X 0,Y 340.723,Z 542.045,A -85,B 0,C 180,E1 -14255.279,E2 -14255.279} C_VEL
LIN {X 0,Y 340.716,Z 542.04,A -85,B 0,C 180,E1 -14258.386,E2 -14258.386} C_VEL
LIN {X 0,Y 340.702,Z 541.998,A -85,B 0,C 180,E1 -14262.045,E2 -14262.045} C_VEL
LIN {X 0,Y 340.656,Z 542.05,A -85,B 0,C 180,E1 -14266.227,E2 -14266.227} C_VEL
LIN {X 0,Y 340.691,Z 542.015,A -85,B 0,C 180,E1 -14269.753,E2 -14269.753} C_VEL
LIN {X 0,Y 340.709,Z 542.046,A -85,B 0,C 180,E1 -14273.258,E2 -14273.258} C_VEL
LIN {X 0,Y 340.696,Z 542.039,A -85,B 0,C 180,E1 -14276.153,E2 -14276.153} C_VEL
LIN {X 0,Y 340.746,Z 542.043,A -85,B 0,C 180,E1 -14280.329,E2 -14280.329} C_VEL
LIN {X 0,Y 340.848,Z 542.17,A -85,B 0,C 180,E1 -14283.106,E2 -14283.106} C_VEL
LIN {X 0,Y 342.923,Z 552.515,A -85,B 0,C 180,E1 -14286.407,E2 -14286.407} C_VEL
LIN {X 0,Y 343.308,Z 553.927,A -85,B 0,C 180,E1 -14286.558,E2 -14286.558} C_VEL
LIN {X 0,Y 347.609,Z 565.505,A -85,B 0,C 180,E1 -14287.132,E2 -14287.132} C_VEL
LIN {X 0,Y 350.803,Z 581.087,A -85,B 0,C 180,E1 -14287.693,E2 -14287.693} C_VEL
LIN {X 0,Y 349.273,Z 659.087,A -85,B 0,C 180,E1 -14289.304,E2 -14289.304} C_VEL
LIN {X 0,Y 348.736,Z 671.757,A -85,B 0,C 180,E1 -14289.772,E2 -14289.772} C_VEL
LIN {X 0,Y 347.922,Z 684.165,A -85,B 0,C 180,E1 -14290.453,E2 -14290.453} C_VEL
LIN {X 0,Y 346.846,Z 696.622,A -85,B 0,C 180,E1 -14291.388,E2 -14291.388} C_VEL
LIN {X 0,Y 345.587,Z 708.53,A -85,B 0,C 180,E1 -14292.574,E2 -14292.574} C_VEL
LIN {X 0,Y 344.566,Z 718.82,A -85,B 0,C 180,E1 -14293.877,E2 -14293.877} C_VEL
LIN {X 0,Y 343.451,Z 727.267,A -85,B 0,C 180,E1 -14295.179,E2 -14295.179} C_VEL
LIN {X 0,Y 342.373,Z 735.137,A -85,B 0,C 180,E1 -14296.647,E2 -14296.647} C_VEL
LIN {X 0,Y 341.341,Z 742.824,A -85,B 0,C 180,E1 -14298.418,E2 -14298.418} C_VEL
LIN {X 0,Y 340.658,Z 748.071,A -85,B 0,C 180,E1 -14299.899,E2 -14299.899} C_VEL
LIN {X 0,Y 339.994,Z 753.163,A -85,B 0,C 180,E1 -14301.679,E2 -14301.679} C_VEL
LIN {X 0,Y 339.638,Z 756.864,A -85,B 0,C 180,E1 -14303.34,E2 -14303.34} C_VEL
LIN {X 0,Y 339.382,Z 760.023,A -85,B 0,C 180,E1 -14305.248,E2 -14305.248} C_VEL
LIN {X 0,Y 339.192,Z 761.423,A -85,B 0,C 180,E1 -14306.435,E2 -14306.435} C_VEL
LIN {X 0,Y 339.063,Z 763.031,A -85,B 0,C 180,E1 -14308.811,E2 -14308.811} C_VEL
LIN {X 0,Y 339.072,Z 763.263,A -85,B 0,C 180,E1 -14309.999,E2 -14309.999} C_VEL
LIN {X 0,Y 339.062,Z 763.074,A -85,B 0,C 180,E1 -14311.187,E2 -14311.187} C_VEL
LIN {X 0,Y 339.187,Z 761.525,A -85,B 0,C 180,E1 -14313.563,E2 -14313.563} C_VEL
LIN {X 0,Y 339.376,Z 760.168,A -85,B 0,C 180,E1 -14314.75,E2 -14314.75} C_VEL
LIN {X 0,Y 339.634,Z 757.082,A -85,B 0,C 180,E1 -14316.655,E2 -14316.655} C_VEL
LIN {X 0,Y 339.991,Z 753.414,A -85,B 0,C 180,E1 -14318.319,E2 -14318.319} C_VEL
LIN {X 0,Y 340.632,Z 748.4,A -85,B 0,C 180,E1 -14320.099,E2 -14320.099} C_VEL
LIN {X 0,Y 341.435,Z 742.086,A -85,B 0,C 180,E1 -14321.877,E2 -14321.877} C_VEL
LIN {X 0,Y 342.457,Z 734.181,A -85,B 0,C 180,E1 -14323.65,E2 -14323.65} C_VEL
LIN {X 0,Y 343.909,Z 724.34,A -85,B 0,C 180,E1 -14325.405,E2 -14325.405} C_VEL
LIN {X 0,Y 345.033,Z 714.022,A -85,B 0,C 180,E1 -14326.872,E2 -14326.872} C_VEL
LIN {X 0,Y 346.245,Z 702.371,A -85,B 0,C 180,E1 -14328.183,E2 -14328.183} C_VEL
LIN {X 0,Y 347.152,Z 693.415,A -85,B 0,C 180,E1 -14328.98,E2 -14328.98} C_VEL
LIN {X 0,Y 347.052,Z 688.138,A -85,B 0,C 180,E1 -14329.419,E2 -14329.419} C_VEL
LIN {X 0,Y 344.989,Z 679.468,A -85,B 0,C 180,E1 -14330.142,E2 -14330.142} C_VEL
LIN {X 0,Y 342.821,Z 670.553,A -85,B 0,C 180,E1 -14330.771,E2 -14330.771} C_VEL
LIN {X 0,Y 342.439,Z 664.894,A -85,B 0,C 180,E1 -14331.04,E2 -14331.04} C_VEL
LIN {X 0,Y 342.96,Z 651.031,A -85,B 0,C 180,E1 -14331.407,E2 -14331.407} C_VEL
LIN {X 0,Y 344.239,Z 581.923,A -85,B 0,C 180,E1 -14332.849,E2 -14332.849} C_VEL
LIN {X 0,Y 340.737,Z 565.77,A -85,B 0,C 180,E1 -14333.463,E2 -14333.463} C_VEL
LIN {X 0,Y 335.875,Z 553.116,A -85,B 0,C 180,E1 -14334.161,E2 -14334.161} C_VEL
LIN {X 0,Y 333.874,Z 543.427,A -85,B 0,C 180,E1 -14337.246,E2 -14337.246} C_VEL
LIN {X 0,Y 333.735,Z 542.919,A -85,B 0,C 180,E1 -14337.598,E2 -14337.598} C_VEL
LIN {X 0,Y 333.688,Z 542.907,A -85,B 0,C 180,E1 -14340.362,E2 -14340.362} C_VEL
LIN {X 0,Y 333.672,Z 542.923,A -85,B 0,C 180,E1 -14344.657,E2 -14344.657} C_VEL
LIN {X 0,Y 333.652,Z 542.926,A -85,B 0,C 180,E1 -14347.649,E2 -14347.649} C_VEL
LIN {X 0,Y 333.647,Z 542.917,A -85,B 0,C 180,E1 -14350.766,E2 -14350.766} C_VEL
LIN {X 0,Y 333.591,Z 542.918,A -85,B 0,C 180,E1 -14354.25,E2 -14354.25} C_VEL
LIN {X 0,Y 333.669,Z 542.924,A -85,B 0,C 180,E1 -14357.622,E2 -14357.622} C_VEL
LIN {X 0,Y 333.673,Z 542.898,A -85,B 0,C 180,E1 -14361.196,E2 -14361.196} C_VEL
LIN {X 0,Y 333.681,Z 542.922,A -85,B 0,C 180,E1 -14365.225,E2 -14365.225} C_VEL
LIN {X 0,Y 333.628,Z 542.922,A -85,B 0,C 180,E1 -14368.221,E2 -14368.221} C_VEL
LIN {X 0,Y 333.705,Z 542.917,A -85,B 0,C 180,E1 -14371.027,E2 -14371.027} C_VEL
LIN {X 0,Y 333.73,Z 542.913,A -85,B 0,C 180,E1 -14373.753,E2 -14373.753} C_VEL
LIN {X 0,Y 333.713,Z 542.906,A -85,B 0,C 180,E1 -14377.913,E2 -14377.913} C_VEL
LIN {X 0,Y 333.787,Z 542.905,A -85,B 0,C 180,E1 -14381.589,E2 -14381.589} C_VEL
LIN {X 0,Y 333.801,Z 542.901,A -85,B 0,C 180,E1 -14385.576,E2 -14385.576} C_VEL
LIN {X 0,Y 333.826,Z 542.895,A -85,B 0,C 180,E1 -14389.078,E2 -14389.078} C_VEL
LIN {X 0,Y 334.018,Z 542.875,A -85,B 0,C 180,E1 -14392.747,E2 -14392.747} C_VEL
LIN {X 0,Y 333.806,Z 542.902,A -85,B 0,C 180,E1 -14395.169,E2 -14395.169} C_VEL
LIN {X 0,Y 334.1,Z 542.856,A -85,B 0,C 180,E1 -14397.589,E2 -14397.589} C_VEL
LIN {X 0,Y 334.26,Z 542.848,A -85,B 0,C 180,E1 -14400,E2 -14400} C_VEL
LIN {X 0,Y 334.1,Z 542.859,A -85,B 0,C 180,E1 -14402.411,E2 -14402.411} C_VEL
LIN {X 0,Y 334.016,Z 542.878,A -85,B 0,C 180,E1 -14406.039,E2 -14406.039} C_VEL
LIN {X 0,Y 333.977,Z 542.877,A -85,B 0,C 180,E1 -14408.501,E2 -14408.501} C_VEL
LIN {X 0,Y 333.788,Z 542.905,A -85,B 0,C 180,E1 -14412.155,E2 -14412.155} C_VEL
LIN {X 0,Y 333.77,Z 542.898,A -85,B 0,C 180,E1 -14415.887,E2 -14415.887} C_VEL
LIN {X 0,Y 333.79,Z 542.904,A -85,B 0,C 180,E1 -14418.656,E2 -14418.656} C_VEL
LIN {X 0,Y 333.686,Z 542.914,A -85,B 0,C 180,E1 -14422.279,E2 -14422.279} C_VEL
LIN {X 0,Y 333.728,Z 542.905,A -85,B 0,C 180,E1 -14426.247,E2 -14426.247} C_VEL
LIN {X 0,Y 333.683,Z 542.919,A -85,B 0,C 180,E1 -14428.975,E2 -14428.975} C_VEL
LIN {X 0,Y 333.64,Z 542.924,A -85,B 0,C 180,E1 -14432.588,E2 -14432.588} C_VEL
LIN {X 0,Y 333.67,Z 542.899,A -85,B 0,C 180,E1 -14436.14,E2 -14436.14} C_VEL
LIN {X 0,Y 333.642,Z 542.923,A -85,B 0,C 180,E1 -14439.193,E2 -14439.193} C_VEL
LIN {X 0,Y 333.636,Z 542.91,A -85,B 0,C 180,E1 -14442.503,E2 -14442.503} C_VEL
LIN {X 0,Y 333.668,Z 542.916,A -85,B 0,C 180,E1 -14445.969,E2 -14445.969} C_VEL
LIN {X 0,Y 333.698,Z 542.92,A -85,B 0,C 180,E1 -14449.306,E2 -14449.306} C_VEL
LIN {X 0,Y 333.663,Z 542.899,A -85,B 0,C 180,E1 -14453.169,E2 -14453.169} C_VEL
LIN {X 0,Y 333.671,Z 542.919,A -85,B 0,C 180,E1 -14455.343,E2 -14455.343} C_VEL
LIN {X 0,Y 333.711,Z 543.01,A -85,B 0,C 180,E1 -14458.317,E2 -14458.317} C_VEL
LIN {X 0,Y 336.044,Z 553.398,A -85,B 0,C 180,E1 -14461.449,E2 -14461.449} C_VEL
LIN {X 0,Y 337.849,Z 562.706,A -85,B 0,C 180,E1 -14464.099,E2 -14464.099} C_VEL
LIN {X 0,Y 338.032,Z 566.442,A -85,B 0,C 180,E1 -14465.103,E2 -14465.103} C_VEL
LIN {X 0,Y 337.585,Z 570.176,A -85,B 0,C 180,E1 -14465.997,E2 -14465.997} C_VEL
LIN {X 0,Y 339.366,Z 579.977,A -85,B 0,C 180,E1 -14466.396,E2 -14466.396} C_VEL
LIN {X 0,Y 343.754,Z 606.691,A -85,B 0,C 180,E1 -14467.305,E2 -14467.305} C_VEL
LIN {X 0,Y 342.399,Z 678.456,A -85,B 0,C 180,E1 -14468.832,E2 -14468.832} C_VEL
LIN {X 0,Y 341.625,Z 691.638,A -85,B 0,C 180,E1 -14469.334,E2 -14469.334} C_VEL
LIN {X 0,Y 340.674,Z 703.76,A -85,B 0,C 180,E1 -14470.022,E2 -14470.022} C_VEL
LIN {X 0,Y 339.445,Z 716.004,A -85,B 0,C 180,E1 -14470.969,E2 -14470.969} C_VEL
LIN {X 0,Y 338.095,Z 727.584,A -85,B 0,C 180,E1 -14472.146,E2 -14472.146} C_VEL
LIN {X 0,Y 336.794,Z 737.975,A -85,B 0,C 180,E1 -14473.478,E2 -14473.478} C_VEL
LIN {X 0,Y 335.739,Z 746.546,A -85,B 0,C 180,E1 -14474.833,E2 -14474.833} C_VEL
LIN {X 0,Y 334.705,Z 754.418,A -85,B 0,C 180,E1 -14476.337,E2 -14476.337} C_VEL
LIN {X 0,Y 333.601,Z 762.106,A -85,B 0,C 180,E1 -14478.148,E2 -14478.148} C_VEL
LIN {X 0,Y 333.007,Z 767.379,A -85,B 0,C 180,E1 -14479.667,E2 -14479.667} C_VEL
LIN {X 0,Y 332.478,Z 772.489,A -85,B 0,C 180,E1 -14481.492,E2 -14481.492} C_VEL
LIN {X 0,Y 332.107,Z 776.461,A -85,B 0,C 180,E1 -14483.317,E2 -14483.317} C_VEL
LIN {X 0,Y 331.981,Z 779.399,A -85,B 0,C 180,E1 -14485.143,E2 -14485.143} C_VEL
LIN {X 0,Y 331.996,Z 780.797,A -85,B 0,C 180,E1 -14486.36,E2 -14486.36} C_VEL
LIN {X 0,Y 331.913,Z 783.923,A -85,B 0,C 180,E1 -14490.001,E2 -14490.001} C_VEL
LIN {X 0,Y 331.883,Z 784.379,A -85,B 0,C 180,E1 -14491.214,E2 -14491.214} C_VEL
LIN {X 0,Y 331.914,Z 784.304,A -85,B 0,C 180,E1 -14492.428,E2 -14492.428} C_VEL
LIN {X 0,Y 332.011,Z 783.697,A -85,B 0,C 180,E1 -14493.642,E2 -14493.642} C_VEL
LIN {X 0,Y 332.079,Z 782.554,A -85,B 0,C 180,E1 -14494.857,E2 -14494.857} C_VEL
LIN {X 0,Y 332.245,Z 779.649,A -85,B 0,C 180,E1 -14496.682,E2 -14496.682} C_VEL
LIN {X 0,Y 332.613,Z 775.449,A -85,B 0,C 180,E1 -14498.507,E2 -14498.507} C_VEL
LIN {X 0,Y 333.162,Z 769.75,A -85,B 0,C 180,E1 -14500.33,E2 -14500.33} C_VEL
LIN {X 0,Y 333.726,Z 763.509,A -85,B 0,C 180,E1 -14501.85,E2 -14501.85} C_VEL
LIN {X 0,Y 335.727,Z 746.447,A -85,B 0,C 180,E1 -14505.17,E2 -14505.17} C_VEL
LIN {X 0,Y 337.012,Z 735.853,A -85,B 0,C 180,E1 -14506.804,E2 -14506.804} C_VEL
LIN {X 0,Y 338.398,Z 724.82,A -85,B 0,C 180,E1 -14508.152,E2 -14508.152} C_VEL
LIN {X 0,Y 339.615,Z 714.119,A -85,B 0,C 180,E1 -14509.18,E2 -14509.18} C_VEL
LIN {X 0,Y 340.864,Z 701.243,A -85,B 0,C 180,E1 -14510.126,E2 -14510.126} C_VEL
LIN {X 0,Y 341.851,Z 688.133,A -85,B 0,C 180,E1 -14510.811,E2 -14510.811} C_VEL
LIN {X 0,Y 342.496,Z 674.994,A -85,B 0,C 180,E1 -14511.243,E2 -14511.243} C_VEL
LIN {X 0,Y 343.711,Z 606.842,A -85,B 0,C 180,E1 -14512.677,E2 -14512.677} C_VEL
LIN {X 0,Y 342.756,Z 599.876,A -85,B 0,C 180,E1 -14512.929,E2 -14512.929} C_VEL
LIN {X 0,Y 343.466,Z 584.393,A -85,B 0,C 180,E1 -14514.48,E2 -14514.48} C_VEL
LIN {X 0,Y 342.767,Z 573.042,A -85,B 0,C 180,E1 -14516.026,E2 -14516.026} C_VEL
LIN {X 0,Y 341.1,Z 564.586,A -85,B 0,C 180,E1 -14517.629,E2 -14517.629} C_VEL
LIN {X 0,Y 339.114,Z 556.902,A -85,B 0,C 180,E1 -14519.491,E2 -14519.491} C_VEL
LIN {X 0,Y 338.009,Z 552.167,A -85,B 0,C 180,E1 -14520.83,E2 -14520.83} C_VEL
LIN {X 0,Y 337.51,Z 550.578,A -85,B 0,C 180,E1 -14521.378,E2 -14521.378} C_VEL
LIN {X 0,Y 335.635,Z 547.019,A -85,B 0,C 180,E1 -14523.115,E2 -14523.115} C_VEL
LIN {X 0,Y 334.056,Z 544.505,A -85,B 0,C 180,E1 -14524.865,E2 -14524.865} C_VEL
LIN {X 0,Y 333.681,Z 543.105,A -85,B 0,C 180,E1 -14525.953,E2 -14525.953} C_VEL
LIN {X 0,Y 333.65,Z 542.923,A -85,B 0,C 180,E1 -14529.193,E2 -14529.193} C_VEL
LIN {X 0,Y 333.636,Z 542.923,A -85,B 0,C 180,E1 -14532.5,E2 -14532.5} C_VEL
LIN {X 0,Y 333.649,Z 543.227,A -85,B 0,C 180,E1 -14535.884,E2 -14535.884} C_VEL
LIN {X 0,Y 334.527,Z 545.565,A -85,B 0,C 180,E1 -14537.757,E2 -14537.757} C_VEL
LIN {X 0,Y 335.58,Z 547.055,A -85,B 0,C 180,E1 -14538.934,E2 -14538.934} C_VEL
LIN {X 0,Y 338.675,Z 554.153,A -85,B 0,C 180,E1 -14542.587,E2 -14542.587} C_VEL
LIN {X 0,Y 341.283,Z 561.612,A -85,B 0,C 180,E1 -14545.459,E2 -14545.459} C_VEL
LIN {X 0,Y 343.353,Z 569.014,A -85,B 0,C 180,E1 -14547.847,E2 -14547.847} C_VEL
LIN {X 0,Y 345.045,Z 577.181,A -85,B 0,C 180,E1 -14550.135,E2 -14550.135} C_VEL
LIN {X 0,Y 345.166,Z 581.266,A -85,B 0,C 180,E1 -14551.109,E2 -14551.109} C_VEL
LIN {X 0,Y 342.23,Z 603.177,A -85,B 0,C 180,E1 -14555.524,E2 -14555.524} C_VEL
LIN {X 0,Y 340.619,Z 617.55,A -85,B 0,C 180,E1 -14558.34,E2 -14558.34} C_VEL
LIN {X 0,Y 343.393,Z 631.47,A -85,B 0,C 180,E1 -14559.274,E2 -14559.274} C_VEL
LIN {X 0,Y 344.878,Z 642.695,A -85,B 0,C 180,E1 -14559.895,E2 -14559.895} C_VEL
LIN {X 0,Y 341.888,Z 700.135,A -85,B 0,C 180,E1 -14561.808,E2 -14561.808} C_VEL
LIN {X 0,Y 341.079,Z 710.197,A -85,B 0,C 180,E1 -14562.306,E2 -14562.306} C_VEL
LIN {X 0,Y 340.146,Z 720.797,A -85,B 0,C 180,E1 -14563.031,E2 -14563.031} C_VEL
LIN {X 0,Y 338.888,Z 731.766,A -85,B 0,C 180,E1 -14564.051,E2 -14564.051} C_VEL
LIN {X 0,Y 337.75,Z 740.519,A -85,B 0,C 180,E1 -14565.078,E2 -14565.078} C_VEL
LIN {X 0,Y 336.509,Z 749.682,A -85,B 0,C 180,E1 -14566.411,E2 -14566.411} C_VEL
LIN {X 0,Y 335.404,Z 757.577,A -85,B 0,C 180,E1 -14567.905,E2 -14567.905} C_VEL
LIN {X 0,Y 334.595,Z 762.786,A -85,B 0,C 180,E1 -14569.103,E2 -14569.103} C_VEL
LIN {X 0,Y 333.876,Z 767.136,A -85,B 0,C 180,E1 -14570.305,E2 -14570.305} C_VEL
LIN {X 0,Y 333.104,Z 772.263,A -85,B 0,C 180,E1 -14572.118,E2 -14572.118} C_VEL
LIN {X 0,Y 332.697,Z 775.988,A -85,B 0,C 180,E1 -14573.937,E2 -14573.937} C_VEL
LIN {X 0,Y 332.346,Z 777.676,A -85,B 0,C 180,E1 -14575.148,E2 -14575.148} C_VEL
LIN {X 0,Y 332.09,Z 778.784,A -85,B 0,C 180,E1 -14576.36,E2 -14576.36} C_VEL
LIN {X 0,Y 331.955,Z 779.364,A -85,B 0,C 180,E1 -14577.573,E2 -14577.573} C_VEL
LIN {X 0,Y 331.884,Z 779.423,A -85,B 0,C 180,E1 -14578.787,E2 -14578.787} C_VEL
LIN {X 0,Y 331.884,Z 778.958,A -85,B 0,C 180,E1 -14580,E2 -14580} C_VEL
LIN {X 0,Y 331.877,Z 777.919,A -85,B 0,C 180,E1 -14581.213,E2 -14581.213} C_VEL
LIN {X 0,Y 331.977,Z 775.221,A -85,B 0,C 180,E1 -14583.034,E2 -14583.034} C_VEL
LIN {X 0,Y 332.126,Z 772.721,A -85,B 0,C 180,E1 -14584.247,E2 -14584.247} C_VEL
LIN {X 0,Y 332.163,Z 768.934,A -85,B 0,C 180,E1 -14585.652,E2 -14585.652} C_VEL
LIN {X 0,Y 332.502,Z 763.408,A -85,B 0,C 180,E1 -14587.244,E2 -14587.244} C_VEL
LIN {X 0,Y 332.73,Z 758.001,A -85,B 0,C 180,E1 -14588.503,E2 -14588.503} C_VEL
LIN {X 0,Y 333.097,Z 751.693,A -85,B 0,C 180,E1 -14589.718,E2 -14589.718} C_VEL
LIN {X 0,Y 333.613,Z 743.048,A -85,B 0,C 180,E1 -14591.083,E2 -14591.083} C_VEL
LIN {X 0,Y 334.244,Z 733.16,A -85,B 0,C 180,E1 -14592.292,E2 -14592.292} C_VEL
LIN {X 0,Y 334.678,Z 725.552,A -85,B 0,C 180,E1 -14593.047,E2 -14593.047} C_VEL
LIN {X 0,Y 335.129,Z 716.08,A -85,B 0,C 180,E1 -14593.801,E2 -14593.801} C_VEL
LIN {X 0,Y 335.432,Z 704.739,A -85,B 0,C 180,E1 -14594.484,E2 -14594.484} C_VEL
LIN {X 0,Y 335.918,Z 691.943,A -85,B 0,C 180,E1 -14594.967,E2 -14594.967} C_VEL
LIN {X 0,Y 336.945,Z 638.533,A -85,B 0,C 180,E1 -14596.52,E2 -14596.52} C_VEL
LIN {X 0,Y 334.986,Z 617.139,A -85,B 0,C 180,E1 -14597.238,E2 -14597.238} C_VEL
LIN {X 0,Y 335.841,Z 601.249,A -85,B 0,C 180,E1 -14600.2,E2 -14600.2} C_VEL
LIN {X 0,Y 337.184,Z 581.199,A -85,B 0,C 180,E1 -14603.981,E2 -14603.981} C_VEL
LIN {X 0,Y 338.185,Z 566.024,A -85,B 0,C 180,E1 -14606.853,E2 -14606.853} C_VEL
LIN {X 0,Y 337.411,Z 560.548,A -85,B 0,C 180,E1 -14607.947,E2 -14607.947} C_VEL
LIN {X 0,Y 334.163,Z 545.394,A -85,B 0,C 180,E1 -14611.078,E2 -14611.078} C_VEL
LIN {X 0,Y 333.708,Z 543.05,A -85,B 0,C 180,E1 -14611.608,E2 -14611.608} C_VEL
LIN {X 0,Y 333.69,Z 542.92,A -85,B 0,C 180,E1 -14614.774,E2 -14614.774} C_VEL
LIN {X 0,Y 333.658,Z 542.924,A -85,B 0,C 180,E1 -14617.651,E2 -14617.651} C_VEL
LIN {X 0,Y 333.65,Z 542.889,A -85,B 0,C 180,E1 -14620.767,E2 -14620.767} C_VEL
LIN {X 0,Y 333.597,Z 542.906,A -85,B 0,C 180,E1 -14624.25,E2 -14624.25} C_VEL
LIN {X 0,Y 333.646,Z 542.92,A -85,B 0,C 180,E1 -14627.618,E2 -14627.618} C_VEL
LIN {X 0,Y 333.656,Z 542.894,A -85,B 0,C 180,E1 -14631.202,E2 -14631.202} C_VEL
LIN {X 0,Y 333.68,Z 542.92,A -85,B 0,C 180,E1 -14633.861,E2 -14633.861} C_VEL
LIN {X 0,Y 333.648,Z 542.925,A -85,B 0,C 180,E1 -14637.413,E2 -14637.413} C_VEL
LIN {X 0,Y 333.694,Z 542.916,A -85,B 0,C 180,E1 -14641.025,E2 -14641.025} C_VEL
LIN {X 0,Y 333.794,Z 543.137,A -85,B 0,C 180,E1 -14642.745,E2 -14642.745} C_VEL
LIN {X 0,Y 335.813,Z 552.823,A -85,B 0,C 180,E1 -14645.894,E2 -14645.894} C_VEL
LIN {X 0,Y 336.353,Z 554.576,A -85,B 0,C 180,E1 -14646.058,E2 -14646.058} C_VEL
LIN {X 0,Y 341.278,Z 567.589,A -85,B 0,C 180,E1 -14646.725,E2 -14646.725} C_VEL
LIN {X 0,Y 344.272,Z 583,A -85,B 0,C 180,E1 -14647.284,E2 -14647.284} C_VEL
LIN {X 0,Y 342.665,Z 659.309,A -85,B 0,C 180,E1 -14648.886,E2 -14648.886} C_VEL
LIN {X 0,Y 342.076,Z 671.972,A -85,B 0,C 180,E1 -14649.36,E2 -14649.36} C_VEL
LIN {X 0,Y 341.259,Z 684.377,A -85,B 0,C 180,E1 -14650.056,E2 -14650.056} C_VEL
LIN {X 0,Y 340.137,Z 696.832,A -85,B 0,C 180,E1 -14651.007,E2 -14651.007} C_VEL
LIN {X 0,Y 338.813,Z 708.74,A -85,B 0,C 180,E1 -14652.214,E2 -14652.214} C_VEL
LIN {X 0,Y 337.774,Z 718.749,A -85,B 0,C 180,E1 -14653.503,E2 -14653.503} C_VEL
LIN {X 0,Y 336.582,Z 727.475,A -85,B 0,C 180,E1 -14654.869,E2 -14654.869} C_VEL
LIN {X 0,Y 335.474,Z 735.344,A -85,B 0,C 180,E1 -14656.367,E2 -14656.367} C_VEL
LIN {X 0,Y 334.389,Z 743.03,A -85,B 0,C 180,E1 -14658.174,E2 -14658.174} C_VEL
LIN {X 0,Y 333.666,Z 748.278,A -85,B 0,C 180,E1 -14659.685,E2 -14659.685} C_VEL
LIN {X 0,Y 332.949,Z 753.37,A -85,B 0,C 180,E1 -14661.502,E2 -14661.502} C_VEL
LIN {X 0,Y 332.553,Z 757.368,A -85,B 0,C 180,E1 -14663.354,E2 -14663.354} C_VEL
LIN {X 0,Y 332.304,Z 760.228,A -85,B 0,C 180,E1 -14665.146,E2 -14665.146} C_VEL
LIN {X 0,Y 332.123,Z 761.627,A -85,B 0,C 180,E1 -14666.359,E2 -14666.359} C_VEL
LIN {X 0,Y 331.968,Z 763.236,A -85,B 0,C 180,E1 -14668.786,E2 -14668.786} C_VEL
LIN {X 0,Y 331.975,Z 763.467,A -85,B 0,C 180,E1 -14669.999,E2 -14669.999} C_VEL
LIN {X 0,Y 331.968,Z 763.278,A -85,B 0,C 180,E1 -14671.212,E2 -14671.212} C_VEL
LIN {X 0,Y 332.118,Z 761.728,A -85,B 0,C 180,E1 -14673.639,E2 -14673.639} C_VEL
LIN {X 0,Y 332.298,Z 760.372,A -85,B 0,C 180,E1 -14674.852,E2 -14674.852} C_VEL
LIN {X 0,Y 332.548,Z 757.564,A -85,B 0,C 180,E1 -14676.64,E2 -14676.64} C_VEL
LIN {X 0,Y 332.944,Z 753.618,A -85,B 0,C 180,E1 -14678.496,E2 -14678.496} C_VEL
LIN {X 0,Y 333.642,Z 748.603,A -85,B 0,C 180,E1 -14680.313,E2 -14680.313} C_VEL
LIN {X 0,Y 334.495,Z 742.289,A -85,B 0,C 180,E1 -14682.128,E2 -14682.128} C_VEL
LIN {X 0,Y 335.553,Z 734.383,A -85,B 0,C 180,E1 -14683.936,E2 -14683.936} C_VEL
LIN {X 0,Y 337.083,Z 724.542,A -85,B 0,C 180,E1 -14685.725,E2 -14685.725} C_VEL
LIN {X 0,Y 338.264,Z 714.222,A -85,B 0,C 180,E1 -14687.22,E2 -14687.22} C_VEL
LIN {X 0,Y 339.371,Z 703.992,A -85,B 0,C 180,E1 -14688.409,E2 -14688.409} C_VEL
LIN {X 0,Y 340.561,Z 692.79,A -85,B 0,C 180,E1 -14689.435,E2 -14689.435} C_VEL
LIN {X 0,Y 341.611,Z 680.159,A -85,B 0,C 180,E1 -14690.313,E2 -14690.313} C_VEL
LIN {X 0,Y 342.355,Z 666.595,A -85,B 0,C 180,E1 -14690.974,E2 -14690.974} C_VEL
LIN {X 0,Y 342.439,Z 664.894,A -85,B 0,C 180,E1 -14691.04,E2 -14691.04} C_VEL
LIN {X 0,Y 341.966,Z 661.067,A -85,B 0,C 180,E1 -14691.215,E2 -14691.215} C_VEL
LIN {X 0,Y 336.976,Z 649.095,A -85,B 0,C 180,E1 -14691.857,E2 -14691.857} C_VEL
LIN {X 0,Y 336.489,Z 645.209,A -85,B 0,C 180,E1 -14691.975,E2 -14691.975} C_VEL
LIN {X 0,Y 337.632,Z 582.674,A -85,B 0,C 180,E1 -14693.31,E2 -14693.31} C_VEL
LIN {X 0,Y 334.509,Z 568.131,A -85,B 0,C 180,E1 -14693.877,E2 -14693.877} C_VEL
LIN {X 0,Y 328.731,Z 553.534,A -85,B 0,C 180,E1 -14694.703,E2 -14694.703} C_VEL
LIN {X 0,Y 328.447,Z 552.211,A -85,B 0,C 180,E1 -14695.009,E2 -14695.009} C_VEL
LIN {X 0,Y 326.704,Z 543.961,A -85,B 0,C 180,E1 -14697.821,E2 -14697.821} C_VEL
LIN {X 0,Y 326.589,Z 543.801,A -85,B 0,C 180,E1 -14701.094,E2 -14701.094} C_VEL
LIN {X 0,Y 326.605,Z 543.804,A -85,B 0,C 180,E1 -14704.018,E2 -14704.018} C_VEL
LIN {X 0,Y 326.627,Z 543.797,A -85,B 0,C 180,E1 -14707.238,E2 -14707.238} C_VEL
LIN {X 0,Y 326.578,Z 543.8,A -85,B 0,C 180,E1 -14711.131,E2 -14711.131} C_VEL
LIN {X 0,Y 326.526,Z 543.795,A -85,B 0,C 180,E1 -14714.742,E2 -14714.742} C_VEL
LIN {X 0,Y 326.593,Z 543.802,A -85,B 0,C 180,E1 -14718.157,E2 -14718.157} C_VEL
LIN {X 0,Y 326.639,Z 543.773,A -85,B 0,C 180,E1 -14721.393,E2 -14721.393} C_VEL
LIN {X 0,Y 326.616,Z 543.799,A -85,B 0,C 180,E1 -14724.85,E2 -14724.85} C_VEL
LIN {X 0,Y 326.604,Z 543.796,A -85,B 0,C 180,E1 -14727.455,E2 -14727.455} C_VEL
LIN {X 0,Y 326.655,Z 543.794,A -85,B 0,C 180,E1 -14730.34,E2 -14730.34} C_VEL
LIN {X 0,Y 326.684,Z 543.789,A -85,B 0,C 180,E1 -14734.516,E2 -14734.516} C_VEL
LIN {X 0,Y 326.64,Z 543.787,A -85,B 0,C 180,E1 -14738.545,E2 -14738.545} C_VEL
LIN {X 0,Y 326.737,Z 543.785,A -85,B 0,C 180,E1 -14741.177,E2 -14741.177} C_VEL
LIN {X 0,Y 326.756,Z 543.777,A -85,B 0,C 180,E1 -14745.433,E2 -14745.433} C_VEL
LIN {X 0,Y 326.762,Z 543.776,A -85,B 0,C 180,E1 -14748.839,E2 -14748.839} C_VEL
LIN {X 0,Y 326.972,Z 543.753,A -85,B 0,C 180,E1 -14752.59,E2 -14752.59} C_VEL
LIN {X 0,Y 326.773,Z 543.779,A -85,B 0,C 180,E1 -14755.065,E2 -14755.065} C_VEL
LIN {X 0,Y 327.041,Z 543.735,A -85,B 0,C 180,E1 -14757.537,E2 -14757.537} C_VEL
LIN {X 0,Y 327.211,Z 543.726,A -85,B 0,C 180,E1 -14760,E2 -14760} C_VEL
LIN {X 0,Y 327.041,Z 543.738,A -85,B 0,C 180,E1 -14762.463,E2 -14762.463} C_VEL
LIN {X 0,Y 326.991,Z 543.752,A -85,B 0,C 180,E1 -14766.169,E2 -14766.169} C_VEL
LIN {X 0,Y 326.907,Z 543.758,A -85,B 0,C 180,E1 -14768.655,E2 -14768.655} C_VEL
LIN {X 0,Y 326.731,Z 543.783,A -85,B 0,C 180,E1 -14772.421,E2 -14772.421} C_VEL
LIN {X 0,Y 326.747,Z 543.78,A -85,B 0,C 180,E1 -14774.958,E2 -14774.958} C_VEL
LIN {X 0,Y 326.728,Z 543.784,A -85,B 0,C 180,E1 -14778.84,E2 -14778.84} C_VEL
LIN {X 0,Y 326.614,Z 543.794,A -85,B 0,C 180,E1 -14782.788,E2 -14782.788} C_VEL
LIN {X 0,Y 326.683,Z 543.79,A -85,B 0,C 180,E1 -14785.484,E2 -14785.484} C_VEL
LIN {X 0,Y 326.641,Z 543.797,A -85,B 0,C 180,E1 -14789.661,E2 -14789.661} C_VEL
LIN {X 0,Y 326.613,Z 543.8,A -85,B 0,C 180,E1 -14792.947,E2 -14792.947} C_VEL
LIN {X 0,Y 326.606,Z 543.784,A -85,B 0,C 180,E1 -14795.52,E2 -14795.52} C_VEL
LIN {X 0,Y 326.606,Z 543.8,A -85,B 0,C 180,E1 -14799.228,E2 -14799.228} C_VEL
LIN {X 0,Y 326.588,Z 543.789,A -85,B 0,C 180,E1 -14802.976,E2 -14802.976} C_VEL
LIN {X 0,Y 326.624,Z 543.789,A -85,B 0,C 180,E1 -14807.019,E2 -14807.019} C_VEL
LIN {X 0,Y 326.641,Z 543.779,A -85,B 0,C 180,E1 -14810.767,E2 -14810.767} C_VEL
LIN {X 0,Y 326.611,Z 543.8,A -85,B 0,C 180,E1 -14814.482,E2 -14814.482} C_VEL
LIN {X 0,Y 326.622,Z 543.838,A -85,B 0,C 180,E1 -14817.824,E2 -14817.824} C_VEL
LIN {X 0,Y 328.912,Z 553.821,A -85,B 0,C 180,E1 -14820.947,E2 -14820.947} C_VEL
LIN {X 0,Y 330.852,Z 563.742,A -85,B 0,C 180,E1 -14823.848,E2 -14823.848} C_VEL
LIN {X 0,Y 331.149,Z 567.479,A -85,B 0,C 180,E1 -14824.885,E2 -14824.885} C_VEL
LIN {X 0,Y 330.842,Z 570.107,A -85,B 0,C 180,E1 -14825.491,E2 -14825.491} C_VEL
LIN {X 0,Y 335.506,Z 596.547,A -85,B 0,C 180,E1 -14826.489,E2 -14826.489} C_VEL
LIN {X 0,Y 337.256,Z 609.328,A -85,B 0,C 180,E1 -14826.907,E2 -14826.907} C_VEL
LIN {X 0,Y 335.787,Z 678.264,A -85,B 0,C 180,E1 -14828.394,E2 -14828.394} C_VEL
LIN {X 0,Y 335.004,Z 691.442,A -85,B 0,C 180,E1 -14828.906,E2 -14828.906} C_VEL
LIN {X 0,Y 334.003,Z 703.561,A -85,B 0,C 180,E1 -14829.605,E2 -14829.605} C_VEL
LIN {X 0,Y 332.724,Z 715.803,A -85,B 0,C 180,E1 -14830.57,E2 -14830.57} C_VEL
LIN {X 0,Y 331.326,Z 727.382,A -85,B 0,C 180,E1 -14831.769,E2 -14831.769} C_VEL
LIN {X 0,Y 329.956,Z 737.813,A -85,B 0,C 180,E1 -14833.131,E2 -14833.131} C_VEL
LIN {X 0,Y 328.882,Z 746.343,A -85,B 0,C 180,E1 -14834.508,E2 -14834.508} C_VEL
LIN {X 0,Y 327.799,Z 754.215,A -85,B 0,C 180,E1 -14836.044,E2 -14836.044} C_VEL
LIN {X 0,Y 326.632,Z 761.902,A -85,B 0,C 180,E1 -14837.891,E2 -14837.891} C_VEL
LIN {X 0,Y 325.785,Z 768.997,A -85,B 0,C 180,E1 -14840.063,E2 -14840.063} C_VEL
LIN {X 0,Y 325.287,Z 773.719,A -85,B 0,C 180,E1 -14841.928,E2 -14841.928} C_VEL
LIN {X 0,Y 324.96,Z 777.331,A -85,B 0,C 180,E1 -14843.793,E2 -14843.793} C_VEL
LIN {X 0,Y 324.89,Z 779.195,A -85,B 0,C 180,E1 -14845.037,E2 -14845.037} C_VEL
LIN {X 0,Y 324.9,Z 780.592,A -85,B 0,C 180,E1 -14846.28,E2 -14846.28} C_VEL
LIN {X 0,Y 324.821,Z 783.691,A -85,B 0,C 180,E1 -14850.001,E2 -14850.001} C_VEL
LIN {X 0,Y 324.794,Z 784.262,A -85,B 0,C 180,E1 -14851.241,E2 -14851.241} C_VEL
LIN {X 0,Y 324.836,Z 784.298,A -85,B 0,C 180,E1 -14852.481,E2 -14852.481} C_VEL
LIN {X 0,Y 324.942,Z 783.802,A -85,B 0,C 180,E1 -14853.721,E2 -14853.721} C_VEL
LIN {X 0,Y 325.006,Z 782.742,A -85,B 0,C 180,E1 -14854.963,E2 -14854.963} C_VEL
LIN {X 0,Y 325.202,Z 780.016,A -85,B 0,C 180,E1 -14856.827,E2 -14856.827} C_VEL
LIN {X 0,Y 325.466,Z 777.515,A -85,B 0,C 180,E1 -14858.07,E2 -14858.07} C_VEL
LIN {X 0,Y 325.832,Z 774.33,A -85,B 0,C 180,E1 -14859.311,E2 -14859.311} C_VEL
LIN {X 0,Y 326.463,Z 768.126,A -85,B 0,C 180,E1 -14861.173,E2 -14861.173} C_VEL
LIN {X 0,Y 327.15,Z 761.613,A -85,B 0,C 180,E1 -14862.721,E2 -14862.721} C_VEL
LIN {X 0,Y 328.057,Z 753.483,A -85,B 0,C 180,E1 -14864.264,E2 -14864.264} C_VEL
LIN {X 0,Y 328.855,Z 746.311,A -85,B 0,C 180,E1 -14865.48,E2 -14865.48} C_VEL
LIN {X 0,Y 330.023,Z 736.823,A -85,B 0,C 180,E1 -14866.995,E2 -14866.995} C_VEL
LIN {X 0,Y 331.476,Z 725.93,A -85,B 0,C 180,E1 -14868.385,E2 -14868.385} C_VEL
LIN {X 0,Y 332.73,Z 715.61,A -85,B 0,C 180,E1 -14869.432,E2 -14869.432} C_VEL
LIN {X 0,Y 333.987,Z 703.293,A -85,B 0,C 180,E1 -14870.398,E2 -14870.398} C_VEL
LIN {X 0,Y 335.05,Z 690.315,A -85,B 0,C 180,E1 -14871.133,E2 -14871.133} C_VEL
LIN {X 0,Y 335.802,Z 677.694,A -85,B 0,C 180,E1 -14871.607,E2 -14871.607} C_VEL
LIN {X 0,Y 337.096,Z 607.206,A -85,B 0,C 180,E1 -14873.135,E2 -14873.135} C_VEL
LIN {X 0,Y 336.908,Z 604.919,A -85,B 0,C 180,E1 -14873.27,E2 -14873.27} C_VEL
LIN {X 0,Y 337.988,Z 588.065,A -85,B 0,C 180,E1 -14874.989,E2 -14874.989} C_VEL
LIN {X 0,Y 337.606,Z 577.335,A -85,B 0,C 180,E1 -14876.473,E2 -14876.473} C_VEL
LIN {X 0,Y 337.18,Z 574.049,A -85,B 0,C 180,E1 -14877.049,E2 -14877.049} C_VEL
LIN {X 0,Y 335.779,Z 567.265,A -85,B 0,C 180,E1 -14878.468,E2 -14878.468} C_VEL
LIN {X 0,Y 333.75,Z 558.518,A -85,B 0,C 180,E1 -14880.799,E2 -14880.799} C_VEL
LIN {X 0,Y 332.868,Z 555.444,A -85,B 0,C 180,E1 -14881.86,E2 -14881.86} C_VEL
LIN {X 0,Y 331.127,Z 552.32,A -85,B 0,C 180,E1 -14883.494,E2 -14883.494} C_VEL
LIN {X 0,Y 329.419,Z 548.915,A -85,B 0,C 180,E1 -14885.834,E2 -14885.834} C_VEL
LIN {X 0,Y 327.96,Z 547.165,A -85,B 0,C 180,E1 -14888.423,E2 -14888.423} C_VEL
LIN {X 0,Y 327.592,Z 546.616,A -85,B 0,C 180,E1 -14890.062,E2 -14890.062} C_VEL
LIN {X 0,Y 327.539,Z 546.593,A -85,B 0,C 180,E1 -14891.696,E2 -14891.696} C_VEL
LIN {X 0,Y 328.454,Z 547.849,A -85,B 0,C 180,E1 -14894.92,E2 -14894.92} C_VEL
LIN {X 0,Y 329.323,Z 549.854,A -85,B 0,C 180,E1 -14896.929,E2 -14896.929} C_VEL
LIN {X 0,Y 330.63,Z 552.088,A -85,B 0,C 180,E1 -14898.78,E2 -14898.78} C_VEL
LIN {X 0,Y 333.283,Z 558.568,A -85,B 0,C 180,E1 -14902.3,E2 -14902.3} C_VEL
LIN {X 0,Y 335.626,Z 565.482,A -85,B 0,C 180,E1 -14905.128,E2 -14905.128} C_VEL
LIN {X 0,Y 337.553,Z 572.784,A -85,B 0,C 180,E1 -14907.58,E2 -14907.58} C_VEL
LIN {X 0,Y 339.067,Z 580.696,A -85,B 0,C 180,E1 -14909.883,E2 -14909.883} C_VEL
LIN {X 0,Y 339.099,Z 584.272,A -85,B 0,C 180,E1 -14910.735,E2 -14910.735} C_VEL
LIN {X 0,Y 336.031,Z 605.087,A -85,B 0,C 180,E1 -14915.026,E2 -14915.026} C_VEL
LIN {X 0,Y 334.47,Z 617.707,A -85,B 0,C 180,E1 -14917.545,E2 -14917.545} C_VEL
LIN {X 0,Y 337.465,Z 632.479,A -85,B 0,C 180,E1 -14918.607,E2 -14918.607} C_VEL
LIN {X 0,Y 338.944,Z 643.842,A -85,B 0,C 180,E1 -14919.268,E2 -14919.268} C_VEL
LIN {X 0,Y 335.749,Z 699.604,A -85,B 0,C 180,E1 -14921.187,E2 -14921.187} C_VEL
LIN {X 0,Y 334.854,Z 710.28,A -85,B 0,C 180,E1 -14921.729,E2 -14921.729} C_VEL
LIN {X 0,Y 333.767,Z 721.782,A -85,B 0,C 180,E1 -14922.539,E2 -14922.539} C_VEL
LIN {X 0,Y 332.581,Z 731.184,A -85,B 0,C 180,E1 -14923.425,E2 -14923.425} C_VEL
LIN {X 0,Y 331.371,Z 740.024,A -85,B 0,C 180,E1 -14924.469,E2 -14924.469} C_VEL
LIN {X 0,Y 330.287,Z 747.311,A -85,B 0,C 180,E1 -14925.521,E2 -14925.521} C_VEL
LIN {X 0,Y 329.055,Z 755.807,A -85,B 0,C 180,E1 -14927.041,E2 -14927.041} C_VEL
LIN {X 0,Y 327.886,Z 762.494,A -85,B 0,C 180,E1 -14928.564,E2 -14928.564} C_VEL
LIN {X 0,Y 326.918,Z 767.882,A -85,B 0,C 180,E1 -14930.097,E2 -14930.097} C_VEL
LIN {X 0,Y 326.319,Z 771.349,A -85,B 0,C 180,E1 -14931.329,E2 -14931.329} C_VEL
LIN {X 0,Y 325.825,Z 774.692,A -85,B 0,C 180,E1 -14932.85,E2 -14932.85} C_VEL
LIN {X 0,Y 325.639,Z 776.363,A -85,B 0,C 180,E1 -14933.805,E2 -14933.805} C_VEL
LIN {X 0,Y 325.303,Z 777.992,A -85,B 0,C 180,E1 -14935.042,E2 -14935.042} C_VEL
LIN {X 0,Y 325.028,Z 779.01,A -85,B 0,C 180,E1 -14936.281,E2 -14936.281} C_VEL
LIN {X 0,Y 324.876,Z 779.481,A -85,B 0,C 180,E1 -14937.52,E2 -14937.52} C_VEL
LIN {X 0,Y 324.796,Z 779.427,A -85,B 0,C 180,E1 -14938.76,E2 -14938.76} C_VEL
LIN {X 0,Y 324.792,Z 778.847,A -85,B 0,C 180,E1 -14940,E2 -14940} C_VEL
LIN {X 0,Y 324.789,Z 777.729,A -85,B 0,C 180,E1 -14941.24,E2 -14941.24} C_VEL
LIN {X 0,Y 324.907,Z 774.861,A -85,B 0,C 180,E1 -14943.1,E2 -14943.1} C_VEL
LIN {X 0,Y 325.04,Z 772.233,A -85,B 0,C 180,E1 -14944.34,E2 -14944.34} C_VEL
LIN {X 0,Y 325.165,Z 766.959,A -85,B 0,C 180,E1 -14946.204,E2 -14946.204} C_VEL
LIN {X 0,Y 325.52,Z 761.288,A -85,B 0,C 180,E1 -14947.755,E2 -14947.755} C_VEL
LIN {X 0,Y 325.871,Z 754.025,A -85,B 0,C 180,E1 -14949.309,E2 -14949.309} C_VEL
LIN {X 0,Y 326.411,Z 745.841,A -85,B 0,C 180,E1 -14950.702,E2 -14950.702} C_VEL
LIN {X 0,Y 326.883,Z 736.835,A -85,B 0,C 180,E1 -14951.943,E2 -14951.943} C_VEL
LIN {X 0,Y 327.494,Z 726.769,A -85,B 0,C 180,E1 -14953.022,E2 -14953.022} C_VEL
LIN {X 0,Y 328.031,Z 716.531,A -85,B 0,C 180,E1 -14953.868,E2 -14953.868} C_VEL
LIN {X 0,Y 328.343,Z 706.737,A -85,B 0,C 180,E1 -14954.487,E2 -14954.487} C_VEL
LIN {X 0,Y 328.823,Z 694.289,A -85,B 0,C 180,E1 -14955.02,E2 -14955.02} C_VEL
LIN {X 0,Y 329.907,Z 638.811,A -85,B 0,C 180,E1 -14956.686,E2 -14956.686} C_VEL
LIN {X 0,Y 327.984,Z 617.293,A -85,B 0,C 180,E1 -14957.422,E2 -14957.422} C_VEL
LIN {X 0,Y 328.824,Z 601.882,A -85,B 0,C 180,E1 -14960.323,E2 -14960.323} C_VEL
LIN {X 0,Y 330.223,Z 581.709,A -85,B 0,C 180,E1 -14964.185,E2 -14964.185} C_VEL
LIN {X 0,Y 331.205,Z 567.178,A -85,B 0,C 180,E1 -14966.972,E2 -14966.972} C_VEL
LIN {X 0,Y 330.291,Z 561.022,A -85,B 0,C 180,E1 -14968.224,E2 -14968.224} C_VEL
LIN {X 0,Y 326.683,Z 543.921,A -85,B 0,C 180,E1 -14971.854,E2 -14971.854} C_VEL
LIN {X 0,Y 326.618,Z 543.802,A -85,B 0,C 180,E1 -14975.519,E2 -14975.519} C_VEL
LIN {X 0,Y 326.616,Z 543.788,A -85,B 0,C 180,E1 -14979.227,E2 -14979.227} C_VEL
LIN {X 0,Y 326.579,Z 543.758,A -85,B 0,C 180,E1 -14982.971,E2 -14982.971} C_VEL
LIN {X 0,Y 326.58,Z 543.807,A -85,B 0,C 180,E1 -14987.028,E2 -14987.028} C_VEL
LIN {X 0,Y 326.615,Z 543.767,A -85,B 0,C 180,E1 -14990.773,E2 -14990.773} C_VEL
LIN {X 0,Y 326.616,Z 543.796,A -85,B 0,C 180,E1 -14994.48,E2 -14994.48} C_VEL
LIN {X 0,Y 326.612,Z 543.802,A -85,B 0,C 180,E1 -14997.455,E2 -14997.455} C_VEL
LIN {X 0,Y 326.652,Z 543.799,A -85,B 0,C 180,E1 -15000.339,E2 -15000.339} C_VEL
LIN {X 0,Y 326.73,Z 544.001,A -85,B 0,C 180,E1 -15002.316,E2 -15002.316} C_VEL
LIN {X 0,Y 328.6,Z 552.916,A -85,B 0,C 180,E1 -15005.304,E2 -15005.304} C_VEL
LIN {X 0,Y 329.022,Z 554.369,A -85,B 0,C 180,E1 -15005.473,E2 -15005.473} C_VEL
LIN {X 0,Y 335.126,Z 570.285,A -85,B 0,C 180,E1 -15006.329,E2 -15006.329} C_VEL
LIN {X 0,Y 337.736,Z 583.715,A -85,B 0,C 180,E1 -15006.83,E2 -15006.83} C_VEL
LIN {X 0,Y 336.078,Z 659.531,A -85,B 0,C 180,E1 -15008.452,E2 -15008.452} C_VEL
LIN {X 0,Y 335.461,Z 672.187,A -85,B 0,C 180,E1 -15008.934,E2 -15008.934} C_VEL
LIN {X 0,Y 334.61,Z 684.589,A -85,B 0,C 180,E1 -15009.642,E2 -15009.642} C_VEL
LIN {X 0,Y 333.424,Z 697.043,A -85,B 0,C 180,E1 -15010.61,E2 -15010.61} C_VEL
LIN {X 0,Y 332.065,Z 708.949,A -85,B 0,C 180,E1 -15011.841,E2 -15011.841} C_VEL
LIN {X 0,Y 330.918,Z 719.381,A -85,B 0,C 180,E1 -15013.215,E2 -15013.215} C_VEL
LIN {X 0,Y 329.514,Z 729.375,A -85,B 0,C 180,E1 -15014.853,E2 -15014.853} C_VEL
LIN {X 0,Y 328.145,Z 738.287,A -85,B 0,C 180,E1 -15016.688,E2 -15016.688} C_VEL
LIN {X 0,Y 327.118,Z 745.456,A -85,B 0,C 180,E1 -15018.536,E2 -15018.536} C_VEL
LIN {X 0,Y 326.378,Z 750.294,A -85,B 0,C 180,E1 -15020.079,E2 -15020.079} C_VEL
LIN {X 0,Y 325.765,Z 754.991,A -85,B 0,C 180,E1 -15021.938,E2 -15021.938} C_VEL
LIN {X 0,Y 325.388,Z 758.58,A -85,B 0,C 180,E1 -15023.799,E2 -15023.799} C_VEL
LIN {X 0,Y 325.229,Z 760.434,A -85,B 0,C 180,E1 -15025.04,E2 -15025.04} C_VEL
LIN {X 0,Y 325.056,Z 761.832,A -85,B 0,C 180,E1 -15026.28,E2 -15026.28} C_VEL
LIN {X 0,Y 324.876,Z 763.44,A -85,B 0,C 180,E1 -15028.759,E2 -15028.759} C_VEL
LIN {X 0,Y 324.88,Z 763.672,A -85,B 0,C 180,E1 -15029.999,E2 -15029.999} C_VEL
LIN {X 0,Y 324.876,Z 763.482,A -85,B 0,C 180,E1 -15031.238,E2 -15031.238} C_VEL
LIN {X 0,Y 325.051,Z 761.932,A -85,B 0,C 180,E1 -15033.718,E2 -15033.718} C_VEL
LIN {X 0,Y 325.223,Z 760.576,A -85,B 0,C 180,E1 -15034.958,E2 -15034.958} C_VEL
LIN {X 0,Y 325.449,Z 758.076,A -85,B 0,C 180,E1 -15036.604,E2 -15036.604} C_VEL
LIN {X 0,Y 325.906,Z 753.822,A -85,B 0,C 180,E1 -15038.681,E2 -15038.681} C_VEL
LIN {X 0,Y 326.657,Z 748.806,A -85,B 0,C 180,E1 -15040.536,E2 -15040.536} C_VEL
LIN {X 0,Y 327.567,Z 742.491,A -85,B 0,C 180,E1 -15042.388,E2 -15042.388} C_VEL
LIN {X 0,Y 328.668,Z 734.585,A -85,B 0,C 180,E1 -15044.234,E2 -15044.234} C_VEL
LIN {X 0,Y 330.266,Z 724.743,A -85,B 0,C 180,E1 -15046.058,E2 -15046.058} C_VEL
LIN {X 0,Y 331.495,Z 714.418,A -85,B 0,C 180,E1 -15047.583,E2 -15047.583} C_VEL
LIN {X 0,Y 332.635,Z 704.192,A -85,B 0,C 180,E1 -15048.795,E2 -15048.795} C_VEL
LIN {X 0,Y 333.885,Z 692.988,A -85,B 0,C 180,E1 -15049.84,E2 -15049.84} C_VEL
LIN {X 0,Y 334.984,Z 680.354,A -85,B 0,C 180,E1 -15050.733,E2 -15050.733} C_VEL
LIN {X 0,Y 335.748,Z 666.786,A -85,B 0,C 180,E1 -15051.407,E2 -15051.407} C_VEL
LIN {X 0,Y 336.242,Z 654.679,A -85,B 0,C 180,E1 -15051.776,E2 -15051.776} C_VEL
LIN {X 0,Y 336.489,Z 645.209,A -85,B 0,C 180,E1 -15051.975,E2 -15051.975} C_VEL
LIN {X 0,Y 336.107,Z 639.401,A -85,B 0,C 180,E1 -15052.133,E2 -15052.133} C_VEL
LIN {X 0,Y 331.22,Z 620.712,A -85,B 0,C 180,E1 -15052.911,E2 -15052.911} C_VEL
LIN {X 0,Y 330.595,Z 614.909,A -85,B 0,C 180,E1 -15053.092,E2 -15053.092} C_VEL
LIN {X 0,Y 331.111,Z 583.473,A -85,B 0,C 180,E1 -15053.782,E2 -15053.782} C_VEL
LIN {X 0,Y 328.36,Z 570.769,A -85,B 0,C 180,E1 -15054.295,E2 -15054.295} C_VEL
LIN {X 0,Y 321.585,Z 553.758,A -85,B 0,C 180,E1 -15055.289,E2 -15055.289} C_VEL
LIN {X 0,Y 321.241,Z 552.288,A -85,B 0,C 180,E1 -15055.653,E2 -15055.653} C_VEL
LIN {X 0,Y 319.637,Z 544.818,A -85,B 0,C 180,E1 -15058.281,E2 -15058.281} C_VEL
LIN {X 0,Y 319.53,Z 544.683,A -85,B 0,C 180,E1 -15061.86,E2 -15061.86} C_VEL
LIN {X 0,Y 319.578,Z 544.671,A -85,B 0,C 180,E1 -15065.542,E2 -15065.542} C_VEL
LIN {X 0,Y 319.578,Z 544.677,A -85,B 0,C 180,E1 -15068.006,E2 -15068.006} C_VEL
LIN {X 0,Y 319.525,Z 544.684,A -85,B 0,C 180,E1 -15071.596,E2 -15071.596} C_VEL
LIN {X 0,Y 319.489,Z 544.671,A -85,B 0,C 180,E1 -15075.257,E2 -15075.257} C_VEL
LIN {X 0,Y 319.564,Z 544.677,A -85,B 0,C 180,E1 -15078.393,E2 -15078.393} C_VEL
LIN {X 0,Y 319.578,Z 544.657,A -85,B 0,C 180,E1 -15082.342,E2 -15082.342} C_VEL
LIN {X 0,Y 319.557,Z 544.68,A -85,B 0,C 180,E1 -15085.123,E2 -15085.123} C_VEL
LIN {X 0,Y 319.565,Z 544.676,A -85,B 0,C 180,E1 -15089.057,E2 -15089.057} C_VEL
LIN {X 0,Y 319.603,Z 544.662,A -85,B 0,C 180,E1 -15092.497,E2 -15092.497} C_VEL
LIN {X 0,Y 319.599,Z 544.676,A -85,B 0,C 180,E1 -15095.303,E2 -15095.303} C_VEL
LIN {X 0,Y 319.59,Z 544.664,A -85,B 0,C 180,E1 -15098.047,E2 -15098.047} C_VEL
LIN {X 0,Y 319.682,Z 544.662,A -85,B 0,C 180,E1 -15100.961,E2 -15100.961} C_VEL
LIN {X 0,Y 319.724,Z 544.651,A -85,B 0,C 180,E1 -15105.275,E2 -15105.275} C_VEL
LIN {X 0,Y 319.75,Z 544.641,A -85,B 0,C 180,E1 -15109.873,E2 -15109.873} C_VEL
LIN {X 0,Y 319.926,Z 544.63,A -85,B 0,C 180,E1 -15112.426,E2 -15112.426} C_VEL
LIN {X 0,Y 319.742,Z 544.654,A -85,B 0,C 180,E1 -15114.956,E2 -15114.956} C_VEL
LIN {X 0,Y 319.984,Z 544.613,A -85,B 0,C 180,E1 -15117.482,E2 -15117.482} C_VEL
LIN {X 0,Y 320.162,Z 544.604,A -85,B 0,C 180,E1 -15120,E2 -15120} C_VEL
LIN {X 0,Y 319.985,Z 544.617,A -85,B 0,C 180,E1 -15122.518,E2 -15122.518} C_VEL
LIN {X 0,Y 319.947,Z 544.629,A -85,B 0,C 180,E1 -15126.306,E2 -15126.306} C_VEL
LIN {X 0,Y 319.836,Z 544.639,A -85,B 0,C 180,E1 -15128.848,E2 -15128.848} C_VEL
LIN {X 0,Y 319.677,Z 544.662,A -85,B 0,C 180,E1 -15132.7,E2 -15132.7} C_VEL
LIN {X 0,Y 319.692,Z 544.655,A -85,B 0,C 180,E1 -15135.296,E2 -15135.296} C_VEL
LIN {X 0,Y 319.67,Z 544.666,A -85,B 0,C 180,E1 -15139.255,E2 -15139.255} C_VEL
LIN {X 0,Y 319.564,Z 544.675,A -85,B 0,C 180,E1 -15143.32,E2 -15143.32} C_VEL
LIN {X 0,Y 319.611,Z 544.664,A -85,B 0,C 180,E1 -15146.09,E2 -15146.09} C_VEL
LIN {X 0,Y 319.573,Z 544.677,A -85,B 0,C 180,E1 -15148.935,E2 -15148.935} C_VEL
LIN {X 0,Y 319.525,Z 544.681,A -85,B 0,C 180,E1 -15151.863,E2 -15151.863} C_VEL
LIN {X 0,Y 319.574,Z 544.659,A -85,B 0,C 180,E1 -15155.544,E2 -15155.544} C_VEL
LIN {X 0,Y 319.552,Z 544.668,A -85,B 0,C 180,E1 -15158.011,E2 -15158.011} C_VEL
LIN {X 0,Y 319.549,Z 544.669,A -85,B 0,C 180,E1 -15161.604,E2 -15161.604} C_VEL
LIN {X 0,Y 319.575,Z 544.679,A -85,B 0,C 180,E1 -15165.275,E2 -15165.275} C_VEL
LIN {X 0,Y 319.575,Z 544.677,A -85,B 0,C 180,E1 -15168.721,E2 -15168.721} C_VEL
LIN {X 0,Y 319.579,Z 544.645,A -85,B 0,C 180,E1 -15172.344,E2 -15172.344} C_VEL
LIN {X 0,Y 319.558,Z 544.68,A -85,B 0,C 180,E1 -15175.125,E2 -15175.125} C_VEL
LIN {X 0,Y 319.584,Z 544.79,A -85,B 0,C 180,E1 -15177.401,E2 -15177.401} C_VEL
LIN {X 0,Y 322.042,Z 555.478,A -85,B 0,C 180,E1 -15180.801,E2 -15180.801} C_VEL
LIN {X 0,Y 323.868,Z 564.77,A -85,B 0,C 180,E1 -15183.587,E2 -15183.587} C_VEL
LIN {X 0,Y 324.192,Z 568.983,A -85,B 0,C 180,E1 -15184.771,E2 -15184.771} C_VEL
LIN {X 0,Y 324.128,Z 570.024,A -85,B 0,C 180,E1 -15184.956,E2 -15184.956} C_VEL
LIN {X 0,Y 329.015,Z 597.521,A -85,B 0,C 180,E1 -15186.023,E2 -15186.023} C_VEL
LIN {X 0,Y 330.741,Z 609.144,A -85,B 0,C 180,E1 -15186.425,E2 -15186.425} C_VEL
LIN {X 0,Y 329.202,Z 678.072,A -85,B 0,C 180,E1 -15187.94,E2 -15187.94} C_VEL
LIN {X 0,Y 328.39,Z 691.246,A -85,B 0,C 180,E1 -15188.46,E2 -15188.46} C_VEL
LIN {X 0,Y 327.359,Z 703.363,A -85,B 0,C 180,E1 -15189.173,E2 -15189.173} C_VEL
LIN {X 0,Y 326.037,Z 715.603,A -85,B 0,C 180,E1 -15190.155,E2 -15190.155} C_VEL
LIN {X 0,Y 324.581,Z 727.181,A -85,B 0,C 180,E1 -15191.376,E2 -15191.376} C_VEL
LIN {X 0,Y 323.164,Z 737.611,A -85,B 0,C 180,E1 -15192.766,E2 -15192.766} C_VEL
LIN {X 0,Y 321.987,Z 746.455,A -85,B 0,C 180,E1 -15194.226,E2 -15194.226} C_VEL
LIN {X 0,Y 320.653,Z 755.387,A -85,B 0,C 180,E1 -15196.05,E2 -15196.05} C_VEL
LIN {X 0,Y 319.501,Z 762.82,A -85,B 0,C 180,E1 -15197.939,E2 -15197.939} C_VEL
LIN {X 0,Y 318.744,Z 768.792,A -85,B 0,C 180,E1 -15199.841,E2 -15199.841} C_VEL
LIN {X 0,Y 318.229,Z 773.514,A -85,B 0,C 180,E1 -15201.748,E2 -15201.748} C_VEL
LIN {X 0,Y 317.89,Z 777.126,A -85,B 0,C 180,E1 -15203.655,E2 -15203.655} C_VEL
LIN {X 0,Y 317.804,Z 778.99,A -85,B 0,C 180,E1 -15204.926,E2 -15204.926} C_VEL
LIN {X 0,Y 317.808,Z 780.388,A -85,B 0,C 180,E1 -15206.197,E2 -15206.197} C_VEL
LIN {X 0,Y 317.721,Z 782.25,A -85,B 0,C 180,E1 -15208.734,E2 -15208.734} C_VEL
LIN {X 0,Y 317.73,Z 783.452,A -85,B 0,C 180,E1 -15210.001,E2 -15210.001} C_VEL
LIN {X 0,Y 317.708,Z 784.14,A -85,B 0,C 180,E1 -15211.269,E2 -15211.269} C_VEL
LIN {X 0,Y 317.759,Z 784.3,A -85,B 0,C 180,E1 -15212.536,E2 -15212.536} C_VEL
LIN {X 0,Y 317.853,Z 783.903,A -85,B 0,C 180,E1 -15213.804,E2 -15213.804} C_VEL
LIN {X 0,Y 317.917,Z 782.888,A -85,B 0,C 180,E1 -15215.074,E2 -15215.074} C_VEL
LIN {X 0,Y 318.167,Z 780.38,A -85,B 0,C 180,E1 -15216.979,E2 -15216.979} C_VEL
LIN {X 0,Y 318.604,Z 776.458,A -85,B 0,C 180,E1 -15218.884,E2 -15218.884} C_VEL
LIN {X 0,Y 319.291,Z 771.128,A -85,B 0,C 180,E1 -15220.784,E2 -15220.784} C_VEL
LIN {X 0,Y 320.128,Z 764.092,A -85,B 0,C 180,E1 -15222.683,E2 -15222.683} C_VEL
LIN {X 0,Y 321.096,Z 756.47,A -85,B 0,C 180,E1 -15224.256,E2 -15224.256} C_VEL
LIN {X 0,Y 321.847,Z 749.441,A -85,B 0,C 180,E1 -15225.475,E2 -15225.475} C_VEL
LIN {X 0,Y 324.048,Z 730.759,A -85,B 0,C 180,E1 -15228.167,E2 -15228.167} C_VEL
LIN {X 0,Y 325.459,Z 720.117,A -85,B 0,C 180,E1 -15229.392,E2 -15229.392} C_VEL
LIN {X 0,Y 326.812,Z 708.228,A -85,B 0,C 180,E1 -15230.455,E2 -15230.455} C_VEL
LIN {X 0,Y 327.995,Z 695.856,A -85,B 0,C 180,E1 -15231.281,E2 -15231.281} C_VEL
LIN {X 0,Y 328.937,Z 683.116,A -85,B 0,C 180,E1 -15231.875,E2 -15231.875} C_VEL
LIN {X 0,Y 329.41,Z 669.678,A -85,B 0,C 180,E1 -15232.254,E2 -15232.254} C_VEL
LIN {X 0,Y 330.686,Z 611.632,A -85,B 0,C 180,E1 -15233.527,E2 -15233.527} C_VEL
LIN {X 0,Y 331.171,Z 608.373,A -85,B 0,C 180,E1 -15233.78,E2 -15233.78} C_VEL
LIN {X 0,Y 332.685,Z 589.901,A -85,B 0,C 180,E1 -15235.738,E2 -15235.738} C_VEL
LIN {X 0,Y 332.339,Z 579.083,A -85,B 0,C 180,E1 -15237.354,E2 -15237.354} C_VEL
LIN {X 0,Y 330.999,Z 571.815,A -85,B 0,C 180,E1 -15238.918,E2 -15238.918} C_VEL
LIN {X 0,Y 329.102,Z 562.978,A -85,B 0,C 180,E1 -15241.328,E2 -15241.328} C_VEL
LIN {X 0,Y 328.217,Z 560.243,A -85,B 0,C 180,E1 -15242.366,E2 -15242.366} C_VEL
LIN {X 0,Y 326.46,Z 557.419,A -85,B 0,C 180,E1 -15244.038,E2 -15244.038} C_VEL
LIN {X 0,Y 325.324,Z 554.965,A -85,B 0,C 180,E1 -15245.683,E2 -15245.683} C_VEL
LIN {X 0,Y 324.262,Z 553.485,A -85,B 0,C 180,E1 -15247.364,E2 -15247.364} C_VEL
LIN {X 0,Y 323.261,Z 552.24,A -85,B 0,C 180,E1 -15250.453,E2 -15250.453} C_VEL
LIN {X 0,Y 323.218,Z 552.344,A -85,B 0,C 180,E1 -15252.382,E2 -15252.382} C_VEL
LIN {X 0,Y 323.654,Z 552.971,A -85,B 0,C 180,E1 -15254.227,E2 -15254.227} C_VEL
LIN {X 0,Y 324.326,Z 554.355,A -85,B 0,C 180,E1 -15256.098,E2 -15256.098} C_VEL
LIN {X 0,Y 325.921,Z 557.772,A -85,B 0,C 180,E1 -15259.002,E2 -15259.002} C_VEL
LIN {X 0,Y 327.602,Z 562.129,A -85,B 0,C 180,E1 -15261.528,E2 -15261.528} C_VEL
LIN {X 0,Y 329.562,Z 567.864,A -85,B 0,C 180,E1 -15264.132,E2 -15264.132} C_VEL
LIN {X 0,Y 331.321,Z 574.32,A -85,B 0,C 180,E1 -15266.529,E2 -15266.529} C_VEL
LIN {X 0,Y 332.523,Z 580.242,A -85,B 0,C 180,E1 -15268.426,E2 -15268.426} C_VEL
LIN {X 0,Y 333.264,Z 585.209,A -85,B 0,C 180,E1 -15269.841,E2 -15269.841} C_VEL
LIN {X 0,Y 332.603,Z 590.072,A -85,B 0,C 180,E1 -15270.922,E2 -15270.922} C_VEL
LIN {X 0,Y 329.504,Z 609.84,A -85,B 0,C 180,E1 -15275.087,E2 -15275.087} C_VEL
LIN {X 0,Y 328.511,Z 617.805,A -85,B 0,C 180,E1 -15276.685,E2 -15276.685} C_VEL
LIN {X 0,Y 331.482,Z 632.506,A -85,B 0,C 180,E1 -15277.822,E2 -15277.822} C_VEL
LIN {X 0,Y 333.092,Z 644.326,A -85,B 0,C 180,E1 -15278.566,E2 -15278.566} C_VEL
LIN {X 0,Y 330.148,Z 693.126,A -85,B 0,C 180,E1 -15280.289,E2 -15280.289} C_VEL
LIN {X 0,Y 329.176,Z 706.008,A -85,B 0,C 180,E1 -15280.837,E2 -15280.837} C_VEL
LIN {X 0,Y 328.029,Z 717.369,A -85,B 0,C 180,E1 -15281.578,E2 -15281.578} C_VEL
LIN {X 0,Y 326.795,Z 727.779,A -85,B 0,C 180,E1 -15282.477,E2 -15282.477} C_VEL
LIN {X 0,Y 325.224,Z 738.413,A -85,B 0,C 180,E1 -15283.685,E2 -15283.685} C_VEL
LIN {X 0,Y 324.203,Z 744.99,A -85,B 0,C 180,E1 -15284.6,E2 -15284.6} C_VEL
LIN {X 0,Y 322.973,Z 752.311,A -85,B 0,C 180,E1 -15285.83,E2 -15285.83} C_VEL
LIN {X 0,Y 321.976,Z 758.378,A -85,B 0,C 180,E1 -15287.072,E2 -15287.072} C_VEL
LIN {X 0,Y 320.792,Z 764.63,A -85,B 0,C 180,E1 -15288.628,E2 -15288.628} C_VEL
LIN {X 0,Y 319.681,Z 770.435,A -85,B 0,C 180,E1 -15290.51,E2 -15290.51} C_VEL
LIN {X 0,Y 319.125,Z 773.466,A -85,B 0,C 180,E1 -15291.77,E2 -15291.77} C_VEL
LIN {X 0,Y 318.589,Z 776.737,A -85,B 0,C 180,E1 -15293.667,E2 -15293.667} C_VEL
LIN {X 0,Y 318.239,Z 778.277,A -85,B 0,C 180,E1 -15294.932,E2 -15294.932} C_VEL
LIN {X 0,Y 317.968,Z 779.245,A -85,B 0,C 180,E1 -15296.198,E2 -15296.198} C_VEL
LIN {X 0,Y 317.8,Z 779.604,A -85,B 0,C 180,E1 -15297.465,E2 -15297.465} C_VEL
LIN {X 0,Y 317.711,Z 779.427,A -85,B 0,C 180,E1 -15298.733,E2 -15298.733} C_VEL
LIN {X 0,Y 317.704,Z 778.731,A -85,B 0,C 180,E1 -15300,E2 -15300} C_VEL
LIN {X 0,Y 317.703,Z 777.496,A -85,B 0,C 180,E1 -15301.268,E2 -15301.268} C_VEL
LIN {X 0,Y 317.839,Z 774.494,A -85,B 0,C 180,E1 -15303.169,E2 -15303.169} C_VEL
LIN {X 0,Y 317.955,Z 771.73,A -85,B 0,C 180,E1 -15304.437,E2 -15304.437} C_VEL
LIN {X 0,Y 318.124,Z 766.296,A -85,B 0,C 180,E1 -15306.342,E2 -15306.342} C_VEL
LIN {X 0,Y 318.444,Z 760.39,A -85,B 0,C 180,E1 -15307.929,E2 -15307.929} C_VEL
LIN {X 0,Y 318.853,Z 752.813,A -85,B 0,C 180,E1 -15309.515,E2 -15309.515} C_VEL
LIN {X 0,Y 319.34,Z 745.389,A -85,B 0,C 180,E1 -15310.782,E2 -15310.782} C_VEL
LIN {X 0,Y 319.837,Z 736.294,A -85,B 0,C 180,E1 -15312.049,E2 -15312.049} C_VEL
LIN {X 0,Y 320.479,Z 726.037,A -85,B 0,C 180,E1 -15313.151,E2 -15313.151} C_VEL
LIN {X 0,Y 320.95,Z 716.718,A -85,B 0,C 180,E1 -15313.938,E2 -15313.938} C_VEL
LIN {X 0,Y 321.283,Z 707.04,A -85,B 0,C 180,E1 -15314.57,E2 -15314.57} C_VEL
LIN {X 0,Y 321.777,Z 693.809,A -85,B 0,C 180,E1 -15315.154,E2 -15315.154} C_VEL
LIN {X 0,Y 322.867,Z 639.205,A -85,B 0,C 180,E1 -15316.857,E2 -15316.857} C_VEL
LIN {X 0,Y 320.989,Z 618.192,A -85,B 0,C 180,E1 -15317.579,E2 -15317.579} C_VEL
LIN {X 0,Y 320.972,Z 616.89,A -85,B 0,C 180,E1 -15317.67,E2 -15317.67} C_VEL
LIN {X 0,Y 322.3,Z 595.741,A -85,B 0,C 180,E1 -15321.759,E2 -15321.759} C_VEL
LIN {X 0,Y 323.724,Z 575.272,A -85,B 0,C 180,E1 -15325.734,E2 -15325.734} C_VEL
LIN {X 0,Y 324.191,Z 567.418,A -85,B 0,C 180,E1 -15327.273,E2 -15327.273} C_VEL
LIN {X 0,Y 322.01,Z 556.126,A -85,B 0,C 180,E1 -15329.637,E2 -15329.637} C_VEL
LIN {X 0,Y 319.617,Z 544.798,A -85,B 0,C 180,E1 -15332.108,E2 -15332.108} C_VEL
LIN {X 0,Y 319.564,Z 544.678,A -85,B 0,C 180,E1 -15336.427,E2 -15336.427} C_VEL
LIN {X 0,Y 319.563,Z 544.661,A -85,B 0,C 180,E1 -15339.668,E2 -15339.668} C_VEL
LIN {X 0,Y 319.525,Z 544.641,A -85,B 0,C 180,E1 -15343.46,E2 -15343.46} C_VEL
LIN {X 0,Y 319.558,Z 544.682,A -85,B 0,C 180,E1 -15347.016,E2 -15347.016} C_VEL
LIN {X 0,Y 319.55,Z 544.645,A -85,B 0,C 180,E1 -15350.37,E2 -15350.37} C_VEL
LIN {X 0,Y 319.584,Z 544.672,A -85,B 0,C 180,E1 -15354.457,E2 -15354.457} C_VEL
LIN {X 0,Y 319.534,Z 544.678,A -85,B 0,C 180,E1 -15358.137,E2 -15358.137} C_VEL
LIN {X 0,Y 319.655,Z 544.79,A -85,B 0,C 180,E1 -15361.822,E2 -15361.822} C_VEL
LIN {X 0,Y 321.396,Z 552.954,A -85,B 0,C 180,E1 -15364.662,E2 -15364.662} C_VEL
LIN {X 0,Y 321.698,Z 554.101,A -85,B 0,C 180,E1 -15364.856,E2 -15364.856} C_VEL
LIN {X 0,Y 328.748,Z 571.946,A -85,B 0,C 180,E1 -15365.874,E2 -15365.874} C_VEL
LIN {X 0,Y 331.211,Z 584.264,A -85,B 0,C 180,E1 -15366.353,E2 -15366.353} C_VEL
LIN {X 0,Y 329.486,Z 659.753,A -85,B 0,C 180,E1 -15367.999,E2 -15367.999} C_VEL
LIN {X 0,Y 328.846,Z 672.402,A -85,B 0,C 180,E1 -15368.489,E2 -15368.489} C_VEL
LIN {X 0,Y 327.981,Z 684.801,A -85,B 0,C 180,E1 -15369.212,E2 -15369.212} C_VEL
LIN {X 0,Y 326.75,Z 697.253,A -85,B 0,C 180,E1 -15370.197,E2 -15370.197} C_VEL
LIN {X 0,Y 325.365,Z 708.9,A -85,B 0,C 180,E1 -15371.42,E2 -15371.42} C_VEL
LIN {X 0,Y 324.22,Z 718.638,A -85,B 0,C 180,E1 -15372.712,E2 -15372.712} C_VEL
LIN {X 0,Y 322.903,Z 727.891,A -85,B 0,C 180,E1 -15374.212,E2 -15374.212} C_VEL
LIN {X 0,Y 321.696,Z 735.758,A -85,B 0,C 180,E1 -15375.771,E2 -15375.771} C_VEL
LIN {X 0,Y 320.484,Z 743.444,A -85,B 0,C 180,E1 -15377.653,E2 -15377.653} C_VEL
LIN {X 0,Y 319.396,Z 750.5,A -85,B 0,C 180,E1 -15379.86,E2 -15379.86} C_VEL
LIN {X 0,Y 318.741,Z 755.197,A -85,B 0,C 180,E1 -15381.759,E2 -15381.759} C_VEL
LIN {X 0,Y 318.336,Z 758.785,A -85,B 0,C 180,E1 -15383.661,E2 -15383.661} C_VEL
LIN {X 0,Y 318.157,Z 760.639,A -85,B 0,C 180,E1 -15384.93,E2 -15384.93} C_VEL
LIN {X 0,Y 317.991,Z 762.037,A -85,B 0,C 180,E1 -15386.197,E2 -15386.197} C_VEL
LIN {X 0,Y 317.787,Z 763.645,A -85,B 0,C 180,E1 -15388.732,E2 -15388.732} C_VEL
LIN {X 0,Y 317.788,Z 763.877,A -85,B 0,C 180,E1 -15389.999,E2 -15389.999} C_VEL
LIN {X 0,Y 317.787,Z 763.687,A -85,B 0,C 180,E1 -15391.266,E2 -15391.266} C_VEL
LIN {X 0,Y 317.986,Z 762.136,A -85,B 0,C 180,E1 -15393.801,E2 -15393.801} C_VEL
LIN {X 0,Y 318.151,Z 760.78,A -85,B 0,C 180,E1 -15395.068,E2 -15395.068} C_VEL
LIN {X 0,Y 318.385,Z 758.494,A -85,B 0,C 180,E1 -15396.622,E2 -15396.622} C_VEL
LIN {X 0,Y 318.892,Z 754.025,A -85,B 0,C 180,E1 -15398.873,E2 -15398.873} C_VEL
LIN {X 0,Y 319.683,Z 749.009,A -85,B 0,C 180,E1 -15400.769,E2 -15400.769} C_VEL
LIN {X 0,Y 320.621,Z 742.694,A -85,B 0,C 180,E1 -15402.661,E2 -15402.661} C_VEL
LIN {X 0,Y 321.8,Z 734.787,A -85,B 0,C 180,E1 -15404.545,E2 -15404.545} C_VEL
LIN {X 0,Y 323.44,Z 724.945,A -85,B 0,C 180,E1 -15406.407,E2 -15406.407} C_VEL
LIN {X 0,Y 324.729,Z 714.619,A -85,B 0,C 180,E1 -15407.962,E2 -15407.962} C_VEL
LIN {X 0,Y 325.92,Z 704.392,A -85,B 0,C 180,E1 -15409.197,E2 -15409.197} C_VEL
LIN {X 0,Y 327.223,Z 693.186,A -85,B 0,C 180,E1 -15410.262,E2 -15410.262} C_VEL
LIN {X 0,Y 328.269,Z 681.805,A -85,B 0,C 180,E1 -15411.095,E2 -15411.095} C_VEL
LIN {X 0,Y 329.087,Z 668.804,A -85,B 0,C 180,E1 -15411.78,E2 -15411.78} C_VEL
LIN {X 0,Y 329.682,Z 654.862,A -85,B 0,C 180,E1 -15412.232,E2 -15412.232} C_VEL
LIN {X 0,Y 330.595,Z 614.909,A -85,B 0,C 180,E1 -15413.092,E2 -15413.092} C_VEL
LIN {X 0,Y 329.738,Z 607.223,A -85,B 0,C 180,E1 -15413.335,E2 -15413.335} C_VEL
LIN {X 0,Y 325.153,Z 588.512,A -85,B 0,C 180,E1 -15414.13,E2 -15414.13} C_VEL
LIN {X 0,Y 324.644,Z 584.662,A -85,B 0,C 180,E1 -15414.262,E2 -15414.262} C_VEL
LIN {X 0,Y 322.247,Z 573.446,A -85,B 0,C 180,E1 -15414.726,E2 -15414.726} C_VEL
LIN {X 0,Y 314.972,Z 555.502,A -85,B 0,C 180,E1 -15415.787,E2 -15415.787} C_VEL
LIN {X 0,Y 314.299,Z 553.507,A -85,B 0,C 180,E1 -15415.977,E2 -15415.977} C_VEL
LIN {X 0,Y 312.937,Z 547.284,A -85,B 0,C 180,E1 -15418.138,E2 -15418.138} C_VEL
LIN {X 0,Y 312.56,Z 545.563,A -85,B 0,C 180,E1 -15418.859,E2 -15418.859} C_VEL
LIN {X 0,Y 312.502,Z 545.554,A -85,B 0,C 180,E1 -15422.665,E2 -15422.665} C_VEL
LIN {X 0,Y 312.533,Z 545.546,A -85,B 0,C 180,E1 -15425.949,E2 -15425.949} C_VEL
LIN {X 0,Y 312.509,Z 545.55,A -85,B 0,C 180,E1 -15429.026,E2 -15429.026} C_VEL
LIN {X 0,Y 312.488,Z 545.56,A -85,B 0,C 180,E1 -15432.43,E2 -15432.43} C_VEL
LIN {X 0,Y 312.473,Z 545.551,A -85,B 0,C 180,E1 -15436.03,E2 -15436.03} C_VEL
LIN {X 0,Y 312.496,Z 545.551,A -85,B 0,C 180,E1 -15439.292,E2 -15439.292} C_VEL
LIN {X 0,Y 312.537,Z 545.537,A -85,B 0,C 180,E1 -15442.616,E2 -15442.616} C_VEL
LIN {X 0,Y 312.514,Z 545.554,A -85,B 0,C 180,E1 -15446.31,E2 -15446.31} C_VEL
LIN {X 0,Y 312.54,Z 545.552,A -85,B 0,C 180,E1 -15450.349,E2 -15450.349} C_VEL
LIN {X 0,Y 312.597,Z 545.546,A -85,B 0,C 180,E1 -15454.064,E2 -15454.064} C_VEL
LIN {X 0,Y 312.581,Z 545.538,A -85,B 0,C 180,E1 -15457.528,E2 -15457.528} C_VEL
LIN {X 0,Y 312.631,Z 545.539,A -85,B 0,C 180,E1 -15461.656,E2 -15461.656} C_VEL
LIN {X 0,Y 312.686,Z 545.532,A -85,B 0,C 180,E1 -15465.686,E2 -15465.686} C_VEL
LIN {X 0,Y 312.695,Z 545.52,A -85,B 0,C 180,E1 -15469.641,E2 -15469.641} C_VEL
LIN {X 0,Y 312.864,Z 545.51,A -85,B 0,C 180,E1 -15472.254,E2 -15472.254} C_VEL
LIN {X 0,Y 312.712,Z 545.529,A -85,B 0,C 180,E1 -15474.842,E2 -15474.842} C_VEL
LIN {X 0,Y 312.985,Z 545.492,A -85,B 0,C 180,E1 -15478.713,E2 -15478.713} C_VEL
LIN {X 0,Y 313.114,Z 545.482,A -85,B 0,C 180,E1 -15480,E2 -15480} C_VEL
LIN {X 0,Y 312.931,Z 545.496,A -85,B 0,C 180,E1 -15482.574,E2 -15482.574} C_VEL
LIN {X 0,Y 312.905,Z 545.506,A -85,B 0,C 180,E1 -15486.448,E2 -15486.448} C_VEL
LIN {X 0,Y 312.78,Z 545.517,A -85,B 0,C 180,E1 -15489.049,E2 -15489.049} C_VEL
LIN {X 0,Y 312.629,Z 545.54,A -85,B 0,C 180,E1 -15492.991,E2 -15492.991} C_VEL
LIN {X 0,Y 312.631,Z 545.531,A -85,B 0,C 180,E1 -15495.65,E2 -15495.65} C_VEL
LIN {X 0,Y 312.6,Z 545.545,A -85,B 0,C 180,E1 -15499.709,E2 -15499.709} C_VEL
LIN {X 0,Y 312.539,Z 545.548,A -85,B 0,C 180,E1 -15502.79,E2 -15502.79} C_VEL
LIN {X 0,Y 312.59,Z 545.54,A -85,B 0,C 180,E1 -15505.934,E2 -15505.934} C_VEL
LIN {X 0,Y 312.531,Z 545.554,A -85,B 0,C 180,E1 -15509.651,E2 -15509.651} C_VEL
LIN {X 0,Y 312.514,Z 545.556,A -85,B 0,C 180,E1 -15513.69,E2 -15513.69} C_VEL
LIN {X 0,Y 312.52,Z 545.535,A -85,B 0,C 180,E1 -15517.386,E2 -15517.386} C_VEL
LIN {X 0,Y 312.486,Z 545.558,A -85,B 0,C 180,E1 -15520.71,E2 -15520.71} C_VEL
LIN {X 0,Y 312.519,Z 545.555,A -85,B 0,C 180,E1 -15524.198,E2 -15524.198} C_VEL
LIN {X 0,Y 312.544,Z 545.546,A -85,B 0,C 180,E1 -15527.907,E2 -15527.907} C_VEL
LIN {X 0,Y 312.541,Z 545.521,A -85,B 0,C 180,E1 -15531.909,E2 -15531.909} C_VEL
LIN {X 0,Y 312.504,Z 545.536,A -85,B 0,C 180,E1 -15535.791,E2 -15535.791} C_VEL
LIN {X 0,Y 312.567,Z 545.684,A -85,B 0,C 180,E1 -15536.913,E2 -15536.913} C_VEL
LIN {X 0,Y 315.148,Z 557.047,A -85,B 0,C 180,E1 -15540.621,E2 -15540.621} C_VEL
LIN {X 0,Y 317.09,Z 567.048,A -85,B 0,C 180,E1 -15543.688,E2 -15543.688} C_VEL
LIN {X 0,Y 317.339,Z 569.658,A -85,B 0,C 180,E1 -15544.371,E2 -15544.371} C_VEL
LIN {X 0,Y 320.424,Z 586.151,A -85,B 0,C 180,E1 -15545.07,E2 -15545.07} C_VEL
LIN {X 0,Y 324.173,Z 609.602,A -85,B 0,C 180,E1 -15545.933,E2 -15545.933} C_VEL
LIN {X 0,Y 322.629,Z 677.881,A -85,B 0,C 180,E1 -15547.466,E2 -15547.466} C_VEL
LIN {X 0,Y 321.803,Z 691.051,A -85,B 0,C 180,E1 -15547.997,E2 -15547.997} C_VEL
LIN {X 0,Y 320.742,Z 703.165,A -85,B 0,C 180,E1 -15548.722,E2 -15548.722} C_VEL
LIN {X 0,Y 319.373,Z 715.403,A -85,B 0,C 180,E1 -15549.723,E2 -15549.723} C_VEL
LIN {X 0,Y 317.861,Z 726.98,A -85,B 0,C 180,E1 -15550.967,E2 -15550.967} C_VEL
LIN {X 0,Y 316.359,Z 737.405,A -85,B 0,C 180,E1 -15552.382,E2 -15552.382} C_VEL
LIN {X 0,Y 315.095,Z 746.596,A -85,B 0,C 180,E1 -15553.939,E2 -15553.939} C_VEL
LIN {X 0,Y 313.733,Z 755.184,A -85,B 0,C 180,E1 -15555.736,E2 -15555.736} C_VEL
LIN {X 0,Y 312.532,Z 762.616,A -85,B 0,C 180,E1 -15557.666,E2 -15557.666} C_VEL
LIN {X 0,Y 311.716,Z 768.587,A -85,B 0,C 180,E1 -15559.61,E2 -15559.61} C_VEL
LIN {X 0,Y 311.191,Z 773.31,A -85,B 0,C 180,E1 -15561.56,E2 -15561.56} C_VEL
LIN {X 0,Y 310.821,Z 776.922,A -85,B 0,C 180,E1 -15563.51,E2 -15563.51} C_VEL
LIN {X 0,Y 310.708,Z 778.785,A -85,B 0,C 180,E1 -15564.81,E2 -15564.81} C_VEL
LIN {X 0,Y 310.718,Z 780.183,A -85,B 0,C 180,E1 -15566.11,E2 -15566.11} C_VEL
LIN {X 0,Y 310.637,Z 781.901,A -85,B 0,C 180,E1 -15568.705,E2 -15568.705} C_VEL
LIN {X 0,Y 310.643,Z 783.191,A -85,B 0,C 180,E1 -15570.001,E2 -15570.001} C_VEL
LIN {X 0,Y 310.624,Z 784.013,A -85,B 0,C 180,E1 -15571.298,E2 -15571.298} C_VEL
LIN {X 0,Y 310.685,Z 784.287,A -85,B 0,C 180,E1 -15572.594,E2 -15572.594} C_VEL
LIN {X 0,Y 310.767,Z 783.938,A -85,B 0,C 180,E1 -15573.891,E2 -15573.891} C_VEL
LIN {X 0,Y 310.935,Z 782.235,A -85,B 0,C 180,E1 -15575.997,E2 -15575.997} C_VEL
LIN {X 0,Y 311.429,Z 778.393,A -85,B 0,C 180,E1 -15578.436,E2 -15578.436} C_VEL
LIN {X 0,Y 312.103,Z 773.815,A -85,B 0,C 180,E1 -15580.379,E2 -15580.379} C_VEL
LIN {X 0,Y 312.946,Z 767.534,A -85,B 0,C 180,E1 -15582.32,E2 -15582.32} C_VEL
LIN {X 0,Y 313.7,Z 762.384,A -85,B 0,C 180,E1 -15583.607,E2 -15583.607} C_VEL
LIN {X 0,Y 314.597,Z 756.212,A -85,B 0,C 180,E1 -15584.888,E2 -15584.888} C_VEL
LIN {X 0,Y 315.344,Z 749.669,A -85,B 0,C 180,E1 -15586.024,E2 -15586.024} C_VEL
LIN {X 0,Y 316.167,Z 741.481,A -85,B 0,C 180,E1 -15587.239,E2 -15587.239} C_VEL
LIN {X 0,Y 318.569,Z 721.359,A -85,B 0,C 180,E1 -15589.661,E2 -15589.661} C_VEL
LIN {X 0,Y 319.973,Z 709.953,A -85,B 0,C 180,E1 -15590.744,E2 -15590.744} C_VEL
LIN {X 0,Y 321.178,Z 698.248,A -85,B 0,C 180,E1 -15591.587,E2 -15591.587} C_VEL
LIN {X 0,Y 322.161,Z 685.656,A -85,B 0,C 180,E1 -15592.233,E2 -15592.233} C_VEL
LIN {X 0,Y 322.796,Z 672.822,A -85,B 0,C 180,E1 -15592.651,E2 -15592.651} C_VEL
LIN {X 0,Y 323.983,Z 620.205,A -85,B 0,C 180,E1 -15593.849,E2 -15593.849} C_VEL
LIN {X 0,Y 324.459,Z 615.76,A -85,B 0,C 180,E1 -15594.055,E2 -15594.055} C_VEL
LIN {X 0,Y 325.735,Z 609.365,A -85,B 0,C 180,E1 -15594.575,E2 -15594.575} C_VEL
LIN {X 0,Y 327.408,Z 592.37,A -85,B 0,C 180,E1 -15596.451,E2 -15596.451} C_VEL
LIN {X 0,Y 327.363,Z 583.54,A -85,B 0,C 180,E1 -15597.806,E2 -15597.806} C_VEL
LIN {X 0,Y 326.118,Z 575.965,A -85,B 0,C 180,E1 -15599.459,E2 -15599.459} C_VEL
LIN {X 0,Y 324.486,Z 567.655,A -85,B 0,C 180,E1 -15601.825,E2 -15601.825} C_VEL
LIN {X 0,Y 323.556,Z 565.11,A -85,B 0,C 180,E1 -15602.891,E2 -15602.891} C_VEL
LIN {X 0,Y 321.031,Z 560.508,A -85,B 0,C 180,E1 -15605.904,E2 -15605.904} C_VEL
LIN {X 0,Y 319.733,Z 558.857,A -85,B 0,C 180,E1 -15607.987,E2 -15607.987} C_VEL
LIN {X 0,Y 319.122,Z 558.108,A -85,B 0,C 180,E1 -15609.693,E2 -15609.693} C_VEL
LIN {X 0,Y 318.848,Z 557.853,A -85,B 0,C 180,E1 -15611.46,E2 -15611.46} C_VEL
LIN {X 0,Y 318.952,Z 558.203,A -85,B 0,C 180,E1 -15613.352,E2 -15613.352} C_VEL
LIN {X 0,Y 319.464,Z 559.128,A -85,B 0,C 180,E1 -15615.253,E2 -15615.253} C_VEL
LIN {X 0,Y 320.655,Z 562.023,A -85,B 0,C 180,E1 -15618.177,E2 -15618.177} C_VEL
LIN {X 0,Y 322.122,Z 565.887,A -85,B 0,C 180,E1 -15620.749,E2 -15620.749} C_VEL
LIN {X 0,Y 323.885,Z 571.17,A -85,B 0,C 180,E1 -15623.406,E2 -15623.406} C_VEL
LIN {X 0,Y 325.481,Z 577.282,A -85,B 0,C 180,E1 -15625.847,E2 -15625.847} C_VEL
LIN {X 0,Y 326.655,Z 583.071,A -85,B 0,C 180,E1 -15627.817,E2 -15627.817} C_VEL
LIN {X 0,Y 327.36,Z 588.97,A -85,B 0,C 180,E1 -15629.577,E2 -15629.577} C_VEL
LIN {X 0,Y 324.347,Z 606.178,A -85,B 0,C 180,E1 -15633.324,E2 -15633.324} C_VEL
LIN {X 0,Y 322.604,Z 617.798,A -85,B 0,C 180,E1 -15635.758,E2 -15635.758} C_VEL
LIN {X 0,Y 325.594,Z 632.517,A -85,B 0,C 180,E1 -15636.977,E2 -15636.977} C_VEL
LIN {X 0,Y 327.289,Z 644.683,A -85,B 0,C 180,E1 -15637.816,E2 -15637.816} C_VEL
LIN {X 0,Y 327.204,Z 648.918,A -85,B 0,C 180,E1 -15638,E2 -15638} C_VEL
LIN {X 0,Y 323.65,Z 700.861,A -85,B 0,C 180,E1 -15639.918,E2 -15639.918} C_VEL
LIN {X 0,Y 322.57,Z 711.647,A -85,B 0,C 180,E1 -15640.511,E2 -15640.511} C_VEL
LIN {X 0,Y 321.311,Z 722.615,A -85,B 0,C 180,E1 -15641.344,E2 -15641.344} C_VEL
LIN {X 0,Y 319.976,Z 731.81,A -85,B 0,C 180,E1 -15642.257,E2 -15642.257} C_VEL
LIN {X 0,Y 318.631,Z 740.499,A -85,B 0,C 180,E1 -15643.337,E2 -15643.337} C_VEL
LIN {X 0,Y 317.186,Z 748.669,A -85,B 0,C 180,E1 -15644.58,E2 -15644.58} C_VEL
LIN {X 0,Y 315.657,Z 756.795,A -85,B 0,C 180,E1 -15646.152,E2 -15646.152} C_VEL
LIN {X 0,Y 314.443,Z 763.305,A -85,B 0,C 180,E1 -15647.741,E2 -15647.741} C_VEL
LIN {X 0,Y 313.455,Z 767.601,A -85,B 0,C 180,E1 -15649.013,E2 -15649.013} C_VEL
LIN {X 0,Y 312.727,Z 771.142,A -85,B 0,C 180,E1 -15650.297,E2 -15650.297} C_VEL
LIN {X 0,Y 311.885,Z 775.188,A -85,B 0,C 180,E1 -15652.23,E2 -15652.23} C_VEL
LIN {X 0,Y 311.544,Z 777.123,A -85,B 0,C 180,E1 -15653.524,E2 -15653.524} C_VEL
LIN {X 0,Y 311.179,Z 778.53,A -85,B 0,C 180,E1 -15654.817,E2 -15654.817} C_VEL
LIN {X 0,Y 310.911,Z 779.414,A -85,B 0,C 180,E1 -15656.112,E2 -15656.112} C_VEL
LIN {X 0,Y 310.727,Z 779.721,A -85,B 0,C 180,E1 -15657.407,E2 -15657.407} C_VEL
LIN {X 0,Y 310.629,Z 779.421,A -85,B 0,C 180,E1 -15658.704,E2 -15658.704} C_VEL
LIN {X 0,Y 310.618,Z 778.592,A -85,B 0,C 180,E1 -15660,E2 -15660} C_VEL
LIN {X 0,Y 310.621,Z 777.226,A -85,B 0,C 180,E1 -15661.297,E2 -15661.297} C_VEL
LIN {X 0,Y 310.774,Z 774.1,A -85,B 0,C 180,E1 -15663.241,E2 -15663.241} C_VEL
LIN {X 0,Y 310.871,Z 771.2,A -85,B 0,C 180,E1 -15664.538,E2 -15664.538} C_VEL
LIN {X 0,Y 310.975,Z 766.917,A -85,B 0,C 180,E1 -15666.064,E2 -15666.064} C_VEL
LIN {X 0,Y 311.352,Z 760.799,A -85,B 0,C 180,E1 -15667.784,E2 -15667.784} C_VEL
LIN {X 0,Y 311.726,Z 753.296,A -85,B 0,C 180,E1 -15669.408,E2 -15669.408} C_VEL
LIN {X 0,Y 312.185,Z 745.93,A -85,B 0,C 180,E1 -15670.704,E2 -15670.704} C_VEL
LIN {X 0,Y 312.727,Z 736.94,A -85,B 0,C 180,E1 -15671.998,E2 -15671.998} C_VEL
LIN {X 0,Y 313.335,Z 726.905,A -85,B 0,C 180,E1 -15673.127,E2 -15673.127} C_VEL
LIN {X 0,Y 313.884,Z 716.74,A -85,B 0,C 180,E1 -15674.01,E2 -15674.01} C_VEL
LIN {X 0,Y 314.202,Z 707.067,A -85,B 0,C 180,E1 -15674.657,E2 -15674.657} C_VEL
LIN {X 0,Y 314.713,Z 693.895,A -85,B 0,C 180,E1 -15675.254,E2 -15675.254} C_VEL
LIN {X 0,Y 315.839,Z 639.828,A -85,B 0,C 180,E1 -15677.001,E2 -15677.001} C_VEL
LIN {X 0,Y 313.944,Z 617.627,A -85,B 0,C 180,E1 -15677.801,E2 -15677.801} C_VEL
LIN {X 0,Y 313.958,Z 616.565,A -85,B 0,C 180,E1 -15677.926,E2 -15677.926} C_VEL
LIN {X 0,Y 315.373,Z 594.527,A -85,B 0,C 180,E1 -15682.262,E2 -15682.262} C_VEL
LIN {X 0,Y 316.787,Z 575.627,A -85,B 0,C 180,E1 -15685.987,E2 -15685.987} C_VEL
LIN {X 0,Y 317.139,Z 567.676,A -85,B 0,C 180,E1 -15687.571,E2 -15687.571} C_VEL
LIN {X 0,Y 314.222,Z 553.556,A -85,B 0,C 180,E1 -15690.592,E2 -15690.592} C_VEL
LIN {X 0,Y 312.587,Z 545.699,A -85,B 0,C 180,E1 -15692.342,E2 -15692.342} C_VEL
LIN {X 0,Y 312.541,Z 545.555,A -85,B 0,C 180,E1 -15695.95,E2 -15695.95} C_VEL
LIN {X 0,Y 312.512,Z 545.547,A -85,B 0,C 180,E1 -15699.027,E2 -15699.027} C_VEL
LIN {X 0,Y 312.494,Z 545.507,A -85,B 0,C 180,E1 -15702.431,E2 -15702.431} C_VEL
LIN {X 0,Y 312.462,Z 545.563,A -85,B 0,C 180,E1 -15706.035,E2 -15706.035} C_VEL
LIN {X 0,Y 312.508,Z 545.522,A -85,B 0,C 180,E1 -15709.874,E2 -15709.874} C_VEL
LIN {X 0,Y 312.539,Z 545.553,A -85,B 0,C 180,E1 -15714.05,E2 -15714.05} C_VEL
LIN {X 0,Y 312.508,Z 545.56,A -85,B 0,C 180,E1 -15717.333,E2 -15717.333} C_VEL
LIN {X 0,Y 312.61,Z 545.758,A -85,B 0,C 180,E1 -15721.404,E2 -15721.404} C_VEL
LIN {X 0,Y 314.374,Z 553.726,A -85,B 0,C 180,E1 -15724.179,E2 -15724.179} C_VEL
LIN {X 0,Y 318.02,Z 562.563,A -85,B 0,C 180,E1 -15724.767,E2 -15724.767} C_VEL
LIN {X 0,Y 322.73,Z 575.21,A -85,B 0,C 180,E1 -15725.468,E2 -15725.468} C_VEL
LIN {X 0,Y 324.684,Z 585.816,A -85,B 0,C 180,E1 -15725.88,E2 -15725.88} C_VEL
LIN {X 0,Y 322.936,Z 659.974,A -85,B 0,C 180,E1 -15727.528,E2 -15727.528} C_VEL
LIN {X 0,Y 322.254,Z 672.618,A -85,B 0,C 180,E1 -15728.027,E2 -15728.027} C_VEL
LIN {X 0,Y 321.363,Z 685.013,A -85,B 0,C 180,E1 -15728.763,E2 -15728.763} C_VEL
LIN {X 0,Y 320.264,Z 695.726,A -85,B 0,C 180,E1 -15729.612,E2 -15729.612} C_VEL
LIN {X 0,Y 319.021,Z 706.474,A -85,B 0,C 180,E1 -15730.703,E2 -15730.703} C_VEL
LIN {X 0,Y 317.607,Z 717.207,A -85,B 0,C 180,E1 -15732.084,E2 -15732.084} C_VEL
LIN {X 0,Y 316.374,Z 726.324,A -85,B 0,C 180,E1 -15733.546,E2 -15733.546} C_VEL
LIN {X 0,Y 314.817,Z 735.966,A -85,B 0,C 180,E1 -15735.454,E2 -15735.454} C_VEL
LIN {X 0,Y 313.561,Z 743.651,A -85,B 0,C 180,E1 -15737.376,E2 -15737.376} C_VEL
LIN {X 0,Y 312.397,Z 750.707,A -85,B 0,C 180,E1 -15739.631,E2 -15739.631} C_VEL
LIN {X 0,Y 311.698,Z 755.403,A -85,B 0,C 180,E1 -15741.571,E2 -15741.571} C_VEL
LIN {X 0,Y 311.267,Z 758.991,A -85,B 0,C 180,E1 -15743.517,E2 -15743.517} C_VEL
LIN {X 0,Y 311.09,Z 760.845,A -85,B 0,C 180,E1 -15744.814,E2 -15744.814} C_VEL
LIN {X 0,Y 310.928,Z 762.241,A -85,B 0,C 180,E1 -15746.111,E2 -15746.111} C_VEL
LIN {X 0,Y 310.701,Z 763.849,A -85,B 0,C 180,E1 -15748.703,E2 -15748.703} C_VEL
LIN {X 0,Y 310.698,Z 764.081,A -85,B 0,C 180,E1 -15749.999,E2 -15749.999} C_VEL
LIN {X 0,Y 310.7,Z 763.891,A -85,B 0,C 180,E1 -15751.295,E2 -15751.295} C_VEL
